# B&R Automation Studio project Parker_BMM_ST_V5_3147_V12 (part 27)

#### alarm.c
```c
/********************************************************************
 * COPYRIGHT --  B&R China
 ********************************************************************
 * Program: gAlarm
 * File: gAlarm.c
 * Author: lijianjun
 * Created: March 06, 2013
 ********************************************************************
 * Implementation of program gAlarm --- gAlarm and gImply control
 ********************************************************************/

#include <bur/plctypes.h>
#include <string.h>

#ifdef _DEFAULT_INCLUDES
#include <AsDefault.h>
#endif

#include "defines.h"
#include "edge.h"
#include "keyap2100.h"
//#include "keyap880.h"
#include "pic_id.h"

/* gAlarm text display mode  */
#define	 S$ALARM_TEXT_TOP	      0
#define	 S$ALARM_TEXT_LIST	   1

/**************************************************************************************
** 			       function ALARM type -- warning or alarm  				  			    **
**************************************************************************************/
void AlarmTyp(Alarm_typ * pInst);

/**************************************************************************************
     	        		I N I T U P  O F   T H E   T A S K
**************************************************************************************/
_INIT void alarm_init ( void )
{
	memset(AlarmBit,0,sizeof(AlarmBit));
	memset(OldPBit ,0,sizeof(OldPBit));
	memset(OldNBit ,0,sizeof(OldNBit));

	memset(&gImply,0,sizeof(gImply));

	AlarmCount = 0;
	TimeCounter  = 30;
	iFunction = 1;

	memset(&AlarmBand,1,sizeof(AlarmBand));
	AlarmTyp(&AlarmBand);

}

/**************************************************************************************
        				C Y C L I C   P A R T   O F   T H E   T A S K
**************************************************************************************/

_CYCLIC void alarm_cyclic ( void )
{
	int i,j;
	if(TimeCounter > 0)
	{
		memset(&gAlarm,0,sizeof(gAlarm));
		memset(&LMold.Alarm,0,sizeof(LMold.Alarm));
		memset(&RMold.Alarm,0,sizeof(RMold.Alarm));

		TimeCounter--;
		return;
	}

	pAlarmband = (USINT *)(&AlarmBand);

	gAlarm.batteryLow     = ap880Battery;
	gAlarm.EmergencyStop  = gMachineIn.InstancyStop;

	IsHeat = 0;
	for (i = 0; i<MAX_IDX_CONTRL_ZONES;i++)
	{
		if (1 == gT_Par.Ctl.OnOff[i])
		{
			IsHeat = 1;
			break;
		}
	}

	if(1 == gT_Par.Status.bLow)
	{
		gMachineInfo.ExtrTLow = 1;
		if(1 == IsHeat)
		{
			gAlarm.ScrewTempLow = 1;
		}
		else
		{
			gAlarm.ScrewTempLow = 0;
		}
	}
	else
	{
		gMachineInfo.ExtrTLow = 0;
		gAlarm.ScrewTempLow   = 0;
	}

	gAlarm.ScrewTempHigh	     = gT_Par.Status.bHigh;
	//	if (1==gAlarm.ScrewTempHigh)
	//	{
	//		gMachineOut.HeatPower=0;
	//	}

	if (1==gAlarm.HeatError)
	{
		gMachineOut.HeatPower=0;
	}

	gAlarm.TempFanErr		= gMachineIn.TempFanErr;
	gAlarm.ThermocoupleBroken = gT_Par.Status.bBroken;
	gAlarm.OilPumpFilter  = !gMachineIn.OilPumpFilter ;
	gAlarm.CoolingPumpFilter = !gMachineIn.CoolingPumpFilter;
	gAlarm.TonnageFilter = !gMachineIn.TonnagePumpFilter;
	gAlarm.PneuForceNormal = !gMachineIn.PneuForceNormal ;

	gAlarm.HeatingPowerNormal = !gMachineIn.HeatingPowerNormal;

	gAlarm.OilPumpErr = gMachineIn.OilPumpErr;
//	gAlarm.AirPressureLow = !gMachineIn.LMold.AirPressureLow || !gMachineIn.RMold.AirPressureLow;
	/*20180926 ipis*/
	gAlarm.OilPump1Overload = gMachineIn.OilPump1Overload;
	gAlarm.OilPump2Overload = gMachineIn.OilPump2Overload;
	gAlarm.ParisonMotorOverload = gMachineIn.ParisonPumpMotorErr;
	gAlarm.PlateMotorOverload = gMachineIn.PlateMotorOverload;

	gAlarm.WaterPressureLow = gMachineIn.WaterPressureLow;

	/* -------------- 風壓異常 延時 ----------------*/
	if (1 == gMachineInfo.Auto) //ipis0924
	{
		//		gAlarm.AirPressureLow = gMachineIn.AirPressureLow ;

		if( gMachineIn.LMold.AirPressureLow || gMachineIn.RMold.AirPressureLow)  //owen 20201027
		{
			gMacTimer.AirPressureLowAlarmDly.IN = 1;
			gMacTimer.AirPressureLowAlarmDly.PT = gUserFix_new.AirPressureLowAlarmDlyTime;
			gAlarm.AirPressureLowDly = 1;
			if(1 == gMacTimer.AirPressureLowAlarmDly.Q)
			{
				gAlarm.AirPressureLow = 1;
				gAlarm.AirPressureLowDly = 0;
				gMacTimer.AirPressureLowAlarmDly.IN = 0;
				gMachineInfo.AirPressureLowDlyFlag = 1;
			}

			switch (AirPressureLowStatus)
			{
				case 0:
					gMacTimer.AirPressureLowAlarmDly.IN = 1;
					gMacTimer.AirPressureLowAlarmDly.PT = gUserFix_new.AirPressureLowAlarmDlyTime;
					gAlarm.AirPressureLowDly = 1;
					if(1 == gMacTimer.AirPressureLowAlarmDly.Q)
					{
						gMacTimer.AirPressureLowAlarmDly.IN = 0;
						gAlarm.AirPressureLowDly = 0;
						gAlarm.AirPressureLow = 1;
						gMachineInfo.AirPressureLowDlyFlag = 1;
						StatusDelay = 2;
						AirPressureLowStatus = 10;
					}
					break;
				case 10:
					AlarmSound = 1;
					if(StatusDelay > 0 )StatusDelay--;
					if( 0 == StatusDelay)
					{
						AirPressureLowStatus = 20;
					}
					//reset

					break;
				case 20:

					break;

			}

		}
		else
		{
			gMacTimer.AirPressureLowAlarmDly.IN = 0;
			gAlarm.AirPressureLowDly  = 0;
			AirPressureLowStatus = 0;
		}
	}
	else
	{
		AirPressureLowStatus = 0;
	}

	gAlarm.Voltage24vNormal = !gMachineIn.Voltage24vNormal;
	gAlarm.L_LubricNormal = !gMachineIn.LMold.LubricNormal;
	gAlarm.R_LubricNormal = !gMachineIn.RMold.LubricNormal;

//	if(1 == LMold.Option.RobotTransfer)
//	{
//		gAlarm.ServoTransferErrL = LMold.Robot.Transfer.Error;
//		gAlarm.ServoTransProtectL = LMold.Robot.Transfer.BwHWSwitch | LMold.Robot.Transfer.FwHWSwitch;
//	}
//	else
//	{
//		gAlarm.ServoTransferErrL = 0;
//		gAlarm.ServoTransProtectL = 0;
//	}

	if(1 == LMold.Option.RobotUpDn)
	{
		gAlarm.ServoUpDnErrL = LMold.Robot.UpDn.Error;
		gAlarm.ServoUpDnProtectL  = LMold.Robot.UpDn.BwHWSwitch | LMold.Robot.UpDn.FwHWSwitch;
	}
	else
	{
		gAlarm.ServoUpDnErrL = 0;
		gAlarm.ServoUpDnProtectL = 0;
	}

//	if(1 == RMold.Option.RobotTransfer)
//	{
//		gAlarm.ServoTransferErrR = RMold.Robot.Transfer.Error;
//		gAlarm.ServoTransProtectR = RMold.Robot.Transfer.BwHWSwitch | RMold.Robot.Transfer.FwHWSwitch;
//	}
//	else
//	{
//		gAlarm.ServoTransferErrR = 0;
//		gAlarm.ServoTransProtectR = 0;
//	}

	if(1 == RMold.Option.RobotUpDn)
	{
		gAlarm.ServoUpDnErrR = RMold.Robot.UpDn.Error;
		gAlarm.ServoUpDnProtectR  = RMold.Robot.UpDn.BwHWSwitch | RMold.Robot.UpDn.FwHWSwitch;
	}
	else
	{
		gAlarm.ServoUpDnErrR = 0;
		gAlarm.ServoUpDnProtectR =0;
	}

	gMachineIn.LMold.CarriageLockLimit = ! LMold.Option.Enable;
	if(LMold.Option.Enable == gMachineIn.LMold.CarriageLockLimit)
	{
		gAlarm.CarriageLockL = 1;
	}
	else
	{
		gAlarm.CarriageLockL = 0;
	}

	gMachineIn.RMold.CarriageLockLimit = ! RMold.Option.Enable;
	if(RMold.Option.Enable == gMachineIn.RMold.CarriageLockLimit)
	{
		gAlarm.CarriageLockR = 1;
	}
	else
	{
		gAlarm.CarriageLockR = 0;
	}

	gAlarm.ModuleErr = gPROCESS_info.moduleErr;

	gAlarm.OilPosition = !gMachineIn.OilPositionNormal;

	gAlarm.LubriFilter   = gMachineIn.LubriFilter;
	gAlarm.LubriOverload = gMachineIn.LubriOverload;

	if(0 == gMachineFix.OilCooling.OilTempAlarm)  gMachineFix.OilCooling.OilTempAlarm = 40;
	if(gMachineInfo.OilTemp > gMachineFix.OilCooling.OilTempAlarm)
	{
		gAlarm.OilTempHigh = 1;
	}
	else
	{
		gAlarm.OilTempHigh = 0;
	}

	if(gServoLinear.Current > -32767 && gServoLinear.Current < 32767)
	{
		gAlarm.ParisonLinearBreak = 0;
	}
	else
	{
		gAlarm.ParisonLinearBreak = 1;
	}

	memcpy(&gAlarm.LAlarm,&LMold.Alarm,sizeof(gAlarm.LAlarm));
	memcpy(&gAlarm.RAlarm,&RMold.Alarm,sizeof(gAlarm.RAlarm));

	memcpy(&gAlarm.LHwAlarm,&LMold.HwAlarm,sizeof(gAlarm.LHwAlarm));
	memcpy(&gAlarm.RHwAlarm,&RMold.HwAlarm,sizeof(gAlarm.RHwAlarm));

	memcpy(AlarmBit,&gAlarm,sizeof(gAlarm));

	IsAlarm   = 0;
	IsWarning = 0;

	/* ------------------------ 当前报警 ----------------------------- */

	for(i=0;i<sizeof(gAlarm);i++)
	{
		if(1 == EDGEPOS(AlarmBit[i],OldPBit[i]))
		{
			gMachineInfo.AlarmIndex = i+1;
			if(1 == pAlarmband[i])
			{
				AlarmSound = 1;
			}
		}
		else if((1 == EDGENEG(AlarmBit[i],OldNBit[i]))&&(0 == gAlarm.EmergencyStop))
		{
			gMachineInfo.AlarmIndex  = 0;
			AlarmSound = 0;
		}
		else
		{
			if(1 == AlarmBit[i])
			{
				gMachineInfo.AlarmIndex = i+1;
			}
		}

		OldPBit[i] = AlarmBit[i];
		OldNBit[i] = AlarmBit[i];

		if(1 == AlarmBit[i])
		{
			if(1 == pAlarmband[i])
			{
				IsAlarm = 1;
			}
			else
			{
				IsWarning = 1;
			}
		}
	}/* for(i=0;i<sizeof(gAlarm);i++) */

	AlarmCount ++;

	/* ------------------------- 警报闪动图标 ---------------------------- */
	if(1 == IsAlarm || 1 == IsWarning)
	{
		if((AlarmCount%10) < 5)
		{
			gMachineInfo.IsAlarm = 1;
		}
		else
		{
			gMachineInfo.IsAlarm = 0;
		}
	}
	else
	{
		gMachineInfo.IsAlarm = 0;
	}

	/* ------------------------- 输出警报文字 ---------------------------- */
	if (gPanelObj.vcHandle == 0)
	{

	}
	else if (IsAlarm || IsWarning)
	{
		if((AlarmCount%3) == 0)
		{
			if (!VA_Saccess (1, gPanelObj.vcHandle))
			{
				if(iFunction > 2 || iFunction < 1)iFunction = 1;
				AlarmLength = sizeof(sAlarmText)/sizeof(sAlarmText[0]);
				Status_wcGetAlarmList = VA_wcGetActAlarmList(1, gPanelObj.vcHandle, (UDINT)sAlarmTmp, (UDINT)&AlarmLength, iFunction, '|', 2);

				if (Status_wcGetAlarmList == 240)
				{
					iFunction = 1;
					lengthTotal = record;
					record = 0;
					memcpy(sAlarmTotal,sAlarmTotalTmp,sizeof(sAlarmTotalTmp));
				}
				else if(Status_wcGetAlarmList == 0)
				{
					if(S$ALARM_TEXT_TOP == gMachineFix.Option.AlarmTextMode )
						{
						iFunction = 1;
					}
					else
					{
						iFunction = 2;
					}

					if(iFunctionOld == 1 && iFunction == 2)
					{
						memset(sAlarmTotalTmp,0,sizeof(sAlarmTotalTmp));
					}

					j = 0;
					for(i=0;i<sizeof(sAlarmText)/sizeof(sAlarmText[0]);i++)
					{
						if(sAlarmTmp[i] == '|')
						{
							IndexArray[j] = i;
							j++;
						}

						if(sAlarmTmp[i] == 0)
						{
							break;
						}
					}/* for(i=0;i<sizeof(sAlarmText)/sizeof(sAlarmText[0]);i++) */

					memset(sAlarmText,0,sizeof(sAlarmText));
					if(IndexArray[3] > IndexArray[2] + 2)
					{
						for(i=IndexArray[2]+1;i<IndexArray[3];i++)
						{
							sAlarmText[i - IndexArray[2] - 1] = sAlarmTmp[i];
							if(record < 180)
							{
								sAlarmTotalTmp[record + i - IndexArray[2] - 1] = sAlarmTmp[i];
							}
						}

						sAlarmTmp[IndexArray[3] - IndexArray[2] - 1] = 0;

						if(record < 180)
						{
							sAlarmTotalTmp[record + IndexArray[3] - IndexArray[2] - 1] = '/';
							record = record + IndexArray[3] - IndexArray[2];
						}
					}/* if(IndexArray[1] > IndexArray[2] + 2) */
				}/* else if(Status_wcGetAlarmList == 0) */
				VA_Srelease (1, gPanelObj.vcHandle);
			}/* if (!VA_Saccess (1, vcHandle)) */
		}/* if((AlarmCount%3) == 0) */
	}
	else  /* else if (IsAlarm) */
	{
		memset(sAlarmText,0,sizeof(sAlarmText));
	}/* if (vcHandle == 0) */

	iFunctionOld = iFunction;

	/* ------------ gAlarm led mode ----------- */

	if (1 == IsAlarm )
	{
		if( 1 == gAlarm.AirPressureLowDly )
		{
			gMachineInfo.AlarmLight.Red = 0;
			gMachineInfo.AlarmLight.Yellow = 1;
			gMachineInfo.AlarmLight.Green = 0;
		}
		else
		{
			gMachineInfo.AlarmLight.Red = 1;
			gMachineInfo.AlarmLight.Yellow = 0;
			gMachineInfo.AlarmLight.Green = 0;
		}
	}
	else
	{
		gMachineInfo.AlarmLight.Red = 0;
		if(1 == gMachineInfo.IsImply ||  (1 == gExtruderTempLow_HMIFlag && 1 == gMachineOut.HeatPower) ) // 加溫啟動 但溫度未到（與壓出機啟動條件相同）
		{
			gMachineInfo.AlarmLight.Yellow = 1;
			gMachineInfo.AlarmLight.Green = 0;
		}
		else
		{
			gMachineInfo.AlarmLight.Yellow = 0;
			gMachineInfo.AlarmLight.Green = 1;
		}

	}

	gMachineOut.AlarmRed 	= gMachineInfo.AlarmLight.Red;
	gMachineOut.AlarmYellow = gMachineInfo.AlarmLight.Yellow;
	gMachineOut.AlarmGreen 	= gMachineInfo.AlarmLight.Green;

	//	if(0 == gMachineFix.Option.AlarmLedMode)
	//	{
	//		gMachineOut.AlarmRed = IsAlarm;
	//	}
	//	else
	//	{
	//		gMachineOut.AlarmRed = gMachineInfo.IsAlarm;
	//	}

	//	gMachineOut.AlarmYellow = IsWarning;

	/* ------------ gAlarm sound mode ----------- */

	if(1 == AlarmSound)
	{
//		if((AlarmCount%8) < 4)
//		{
//			gMachineOut.AlarmBuzzer = 1;
//		}
//		else
//		{
//			gMachineOut.AlarmBuzzer = 0;
//		}

		//Alarm Buzzer Echo Mode
		AlarmBuzzerCount ++;
		if((AlarmBuzzerCount < 5))
		{
			gMachineOut.AlarmBuzzer = 1;
		}
		else
		{
			if(AlarmBuzzerCount > 7) AlarmBuzzerCount = 0;
			gMachineOut.AlarmBuzzer = 0;
		}

//		gMachineOut.AlarmBuzzer = 1;

	}
	else
	{
		gMachineOut.AlarmBuzzer  = 0;
		AlarmBuzzerCount = 0;
	}
	/* ------------------------ 消除报警 -------------------------------- */
	if(1 == EDGEPOS(gPanelObj.KeyMatric[S$KEYMATRIX_ALARM_RESET],OldAlarmConfirmOK))
	{
		memset(&gAlarm,0,sizeof(gAlarm));
		memset(&LMold.Alarm,0,sizeof(LMold.Alarm));
		memset(&RMold.Alarm,0,sizeof(RMold.Alarm));
		memset(&LMold.HwAlarm,0,sizeof(LMold.HwAlarm));
		memset(&RMold.HwAlarm,0,sizeof(RMold.HwAlarm));
		/*gExtruderACtrl.InverterCmd.bResetFault = 1*/
	}

	if(1 == gPanelObj.KeyMatric[S$KEYMATRIX_ALARM_RESET])
	{
		AlarmSound = 0;
		gPROCESS_info.extruderStopEnable = 0;
	}
	OldAlarmConfirmOK = gPanelObj.KeyMatric[S$KEYMATRIX_ALARM_RESET];

	/*Albert P84 Error reset by Visual Key*/
	gExtruderACtrl.InverterCmd.bResetFault = gPanelObj.KeyMatric[S$KEYMATRIX_ALARM_RESET];
	gExtruderBCtrl.InverterCmd.bResetFault = gPanelObj.KeyMatric[S$KEYMATRIX_ALARM_RESET];
	gExtruderCCtrl.InverterCmd.bResetFault = gPanelObj.KeyMatric[S$KEYMATRIX_ALARM_RESET];
	gExtruderVCtrl.InverterCmd.bResetFault = gPanelObj.KeyMatric[S$KEYMATRIX_ALARM_RESET];

		/* ------------------------- 系统提示信息  ------------------------- */
		for(i=0;i<sizeof(gImply);i++)
	{
		if((1 == ((USINT *)&gImply)[i]  ) &&
			(0 == ((USINT*)&OldImply)[i]))    /* edge positive */
		{
			gMachineInfo.ImplyTime  = 51;     /*  10 second gImply time */
			gMachineInfo.IsImply    = 1;
			gMachineInfo.ImplyIdex  = i + 1;
		}
		((USINT *)&OldImply)[i] = (( USINT *)&gImply)[i];
	}

	if(gMachineInfo.ImplyTime > 0)
	{
		gMachineInfo.ImplyTime --;
	}

	if(1 == gMachineInfo.ImplyTime)
	{
		memset(&gImply,0,sizeof(gImply));

		gMachineInfo.IsImply   = 0;
		gMachineInfo.ImplyIdex = 0;
	}

	for(i=0;i<32;i++)
	{
		if(1 == gPanelObj.KeyMatric[i] )
		{
			if(1 == gMachineInfo.Manual || 1 == gMachineInfo.Calib )
			{
				if ( 1 == gMachineInfo.IsImply ) gMachineOut.ImplyBuzzer  = 1;
			}
		}

//		if(1 == EDGEPOS(gPanelObj.KeyMatric[i],PKeyMatric[i]) )
//		{
//			if(1 == gMachineInfo.Manual || 1 == gMachineInfo.Calib )
//			{
//				if ( 1 == gMachineInfo.IsImply ) gMachineOut.ImplyBuzzer  = 1;
//			}
//
//		}

		if(1 ==  EDGENEG(gPanelObj.KeyMatric[i],NKeyMatric[i]) )
		{
			gMachineOut.ImplyBuzzer  = 0;
			gMachineInfo.ImplyTime = 2 ;
		}
	}
}/* task end */

void AlarmTyp(Alarm_typ * pInst)
{
	pInst->batteryLow     = 0;
	pInst->ModuleErr      = 1;
	pInst->SaftyDoor      = 1;
	pInst->EmergencyStop  = 1;

	pInst->ScrewTempLow   = 0;
	pInst->ScrewTempHigh  = 0;
	pInst->ThermocoupleBroken = 1;
	pInst->TempException      = 1;

	pInst->OilPumpErr      = 1;
	pInst->CoolingPumpErr  = 0;
	pInst->VisuExtrMotorOverload = 1;
	pInst->A_ExtruderMotorOverload = 1;
	pInst->B_ExtruderMotorOverload = 1;

	pInst->ParisonLinearBreak   = 1;
	pInst->ParisonLinearCalErr  = 1;
	pInst->ParisonValuebeyond   = 0;
	pInst->OilPumpFilter        = 0;

	memset(&pInst->LAlarm,1,sizeof(pInst->LAlarm));
	memset(&pInst->RAlarm,1,sizeof(pInst->RAlarm));
//	pInst->LAlarm.ParisonTimeSmall = 0;
//	pInst->RAlarm.ParisonTimeSmall = 0;

	pInst->LCycleTime = 1;
	pInst->RCycleTime = 1;

	pInst->OilPosition  = 0;
	pInst->LubrTimeZero    = 0;

	pInst->OilTempHigh = 0;
	pInst->OilPumpOff  = 1;

	pInst->LCarriageLinearBreak = 1;
	pInst->RCarriageLinearBreak = 1;
	pInst->LClampLinearBreak = 1;
	pInst->RClampLinearBreak = 1;

	pInst->LowSafeValvePumpOff = 1;
	pInst->HighSafeValvePumpOff = 1;
	pInst->LubriFilter   = 0;
	pInst->LubriOverload = 0;

	pInst->VisuExtrCoolOverload = 0;
	pInst->CoolingPumpErr  = 0;
	pInst->AccuSensorError  = 1;
	pInst->AccuChargeError  = 1;

	pInst->ExtrAMeltP_Alarm  = 1;
	pInst->ExtrBMeltP_Alarm = 1;
	pInst->ExtrACurrentAlarm  = 1;
	pInst->ExtrBCurrentAlarm = 1;
	pInst->A_ExtrMotorOverload =1;
	pInst->B_ExtrMotorOverload =1;
	pInst->C_ExtrMotorOverload =1;
	pInst->V_ExtrMotorOverload =1;

	pInst->HeatError=1;

	pInst->AccuChargeRPressure =1;
	pInst->AirPressureLow = 1;
	pInst->AirPressureLowDly = 1;
	pInst->OilTempHigh	= 1;

	pInst->AirPressureLow=1; //ipis0924
	pInst->WaterPressureLow=1;//ipis0924

}/*  void AlarmTyp(Alarm_typ * pInst) */
```

#### alarm.var
```iecst
VAR
	AlarmBit : ARRAY[0..MAX_ALARM_NUM] OF BOOL;
	AlarmBand : Alarm_typ;
	pAlarmband : REFERENCE TO USINT;
	iFunctionOld : UINT;
	iFunction : UINT;
	Status_wcGetAlarmList : UINT;
	AlarmLength : UINT;
	lengthTotal : UINT;
	record : UINT;
	TimeCounter : UDINT;
	AlarmSound : USINT;
	ImplySound : USINT;
	IsAlarm : USINT;
	IsWarning : USINT;
	OldImply : Imply_typ;
	OldPBit : ARRAY[0..MAX_ALARM_NUM] OF USINT;
	OldNBit : ARRAY[0..MAX_ALARM_NUM] OF USINT;
	OldAlarmConfirmOK : USINT;
	IsHeat : USINT;
	AlarmCount : UDINT;
	ap880Battery : USINT;
	IndexArray : ARRAY[0..9] OF UINT;
	sAlarmText : ARRAY[0..MAX_ALARM_TEXT] OF UINT;
	sAlarmTmp : ARRAY[0..MAX_ALARM_TEXT] OF UINT;
	sAlarmTotalTmp : ARRAY[0..199] OF UINT := [200(0)];
	sAlarmTotal : ARRAY[0..199] OF UINT;
	PKeyMatric : ARRAY[0..MAX_KEY_COUNT] OF USINT;
	NKeyMatric : ARRAY[0..MAX_KEY_COUNT] OF USINT;
	AirPressureLowStatus : UINT;
	StatusDelay : USINT;
	AlarmBuzzerCount : USINT;
END_VAR
```

- pic_id.h (reference to Logical/GlobalIncludes/pic_id.h)

- defines.h (reference to Logical/GlobalIncludes/defines.h)

- keyap880.h (reference to Logical/GlobalIncludes/keyap880.h)

### Program Logical/machine/energy (ANSIC)

#### Variables.var
```iecst
VAR
	tTask : REAL := 0.0;
	RTInfo_v : RTInfo;
	cntRunTime : UDINT;
	tEnergyTime_1 : REAL;
	tEnergyTimeDis_1 : REAL;
	tEnergyTime_2 : REAL;
	tEnergyTimeDis_2 : REAL;
	AvgEnergyOld : REAL;
	AvgEnergyHeatingOld : REAL;
	tEnergyTime_3 : REAL;
	tEnergyTimeDis_3 : REAL;
	AvgEnergyPumpOld : REAL;
END_VAR
```

#### Main.c
```c
#include <bur/plctypes.h>

#ifdef _DEFAULT_INCLUDES
	#include <AsDefault.h>
#endif

void _INIT ProgramInit(void)
{
	// Insert code here
	RTInfo_v.enable = 1;
	RTInfo(&RTInfo_v);
	tTask  = RTInfo_v.cycle_time/1000.0/1000.0;

	tEnergyTime_1 = 0.0;
	tEnergyTime_2 = 0.0;

	cntRunTime = 0;

}

void _CYCLIC ProgramCyclic(void)
{
	// Insert code here
	UDINT  Temp;

	/* ---------------------------- Energy monitor ------------------------- */
	if(gUserPara.SetTimePower < 1)gUserPara.SetTimePower = 10;
	Temp  = (UDINT)(gUserPara.SetTimePower * 60 / tTask);

	if(1 == gMachineInfo.Auto)
	{
		if(cntRunTime >= Temp * 100 )cntRunTime = 0;
		if(0 == (cntRunTime % Temp))
		{
//			gMachineInfo.AvgEnergy = (gMachineInfo.AenergyT_1 - AvgEnergyOld) * 60.0 /gUserPara.SetTimePower;
//			gMachineInfo.AvgEnergyHeating = (gMachineInfo.AenergyT_2 - AvgEnergyHeatingOld)* 60.0 /gUserPara.SetTimePower;

			gMachineInfo.EnergyInfo[0].AvgEnergy = (gMachineInfo.EnergyInfo[0].AenergyT - AvgEnergyOld) * 60.0 /gUserPara.SetTimePower;/*Albert*/
			gMachineInfo.EnergyInfo[1].AvgEnergy = (gMachineInfo.EnergyInfo[1].AenergyT - AvgEnergyHeatingOld)* 60.0 /gUserPara.SetTimePower;/*Albert*/
			gMachineInfo.EnergyInfo[2].AvgEnergy = (gMachineInfo.EnergyInfo[2].AenergyT - AvgEnergyPumpOld) * 60.0/gUserPara.SetTimePower;/*Albert*/

//			AvgEnergyOld = gMachineInfo.AenergyT_1 ;
//			AvgEnergyHeatingOld = gMachineInfo.AenergyT_2 ;

			AvgEnergyOld = gMachineInfo.EnergyInfo[0].AenergyT;
			AvgEnergyHeatingOld = gMachineInfo.EnergyInfo[1].AenergyT;
			AvgEnergyPumpOld = gMachineInfo.EnergyInfo[2].AenergyT;/*Albert for pump consumption*/
		}
		cntRunTime = cntRunTime + 1;
	}
	else
	{
		cntRunTime = 0;
	}

	/* First AP3131 Old*/
	if(1 == gHardWare.AP3131_1.ClearEnergy)
	{
		tEnergyTime_1 = 0.0;
		AvgEnergyOld = 0;/*Albert*/
	}
	else
	{
		tEnergyTime_1 = tEnergyTime_1 + tTask;
	}

	tEnergyTimeDis_1 = tEnergyTime_1/60.0;

	gHardWare.AP3131_1.EnableEnergy = 1;
	if(gUserPara.Current32767_A < 1.0)gUserPara.Current32767_A = 300.0;
	gUserPara.Power32767_A   = 4.0;

	gMachineInfo.Current_A1 = gHardWare.AP3131_1.IrmsA * gUserPara.Current32767_A/1000.0/50.0;
	gMachineInfo.Current_B1 = gHardWare.AP3131_1.IrmsB * gUserPara.Current32767_A/1000.0/50.0;
	gMachineInfo.Current_C1 = gHardWare.AP3131_1.IrmsC * gUserPara.Current32767_A/1000.0/50.0;
	gMachineInfo.Power_1    = gHardWare.AP3131_1.PmeanT * gUserPara.Power32767_A/1000.0;
	gMachineInfo.AenergyT_1 = gHardWare.AP3131_1.AenergyT * gUserPara.Current32767_A/1000.0/50.0;
	gMachineInfo.SumAenergyT_1 = gHardWare.AP3131_1.SAenergyT * gUserPara.Current32767_A/1000.0/50.0;

	/*First AP3131 New*/

	gMachineInfo.EnergyInfo[0].Current_A = gHardWare.AP3131_1.IrmsA * gUserPara.Current32767_A/1000.0/50.0;
	gMachineInfo.EnergyInfo[0].Current_B = gHardWare.AP3131_1.IrmsB * gUserPara.Current32767_A/1000.0/50.0;
	gMachineInfo.EnergyInfo[0].Current_C = gHardWare.AP3131_1.IrmsC * gUserPara.Current32767_A/1000.0/50.0;
	gMachineInfo.EnergyInfo[0].Power    = gHardWare.AP3131_1.PmeanT * gUserPara.Power32767_A/1000.0;
	gMachineInfo.EnergyInfo[0].AenergyT = gHardWare.AP3131_1.AenergyT * gUserPara.Current32767_A/1000.0/50.0;
	gMachineInfo.EnergyInfo[0].SumAenergyT = gHardWare.AP3131_1.SAenergyT * gUserPara.Current32767_A/1000.0/50.0;

	/* Second AP3131 old */
	if(1 == gHardWare.AP3131_2.ClearEnergy)
	{
		tEnergyTime_2 = 0.0;
		AvgEnergyHeatingOld = 0; /*Albert*/
	}
	else
	{
		tEnergyTime_2 = tEnergyTime_2 + tTask;
	}

	tEnergyTimeDis_2 = tEnergyTime_2/60.0;

	gHardWare.AP3131_2.EnableEnergy = 1;
	if(gUserPara.Current32767_B < 1.0)gUserPara.Current32767_B = 100.0;
	gUserPara.Power32767_B = 4.0;

	gMachineInfo.Current_A2 = gHardWare.AP3131_2.IrmsA * gUserPara.Current32767_B/1000.0/50.0;
	gMachineInfo.Current_B2 = gHardWare.AP3131_2.IrmsB * gUserPara.Current32767_B/1000.0/50.0;
	gMachineInfo.Current_C2 = gHardWare.AP3131_2.IrmsC * gUserPara.Current32767_B/1000.0/50.0;
	gMachineInfo.Power_2    = gHardWare.AP3131_2.PmeanT * gUserPara.Power32767_B/1000.0;
	gMachineInfo.AenergyT_2 = gHardWare.AP3131_2.AenergyT * gUserPara.Current32767_B/1000.0/50.0;
	gMachineInfo.SumAenergyT_2 = gHardWare.AP3131_2.SAenergyT * gUserPara.Current32767_B/1000.0/50.0;

	/* Second AP3131 New*/

	gMachineInfo.EnergyInfo[1].Current_A = gHardWare.AP3131_2.IrmsA * gUserPara.Current32767_B/1000.0/50.0;
	gMachineInfo.EnergyInfo[1].Current_B = gHardWare.AP3131_2.IrmsB * gUserPara.Current32767_B/1000.0/50.0;
	gMachineInfo.EnergyInfo[1].Current_C = gHardWare.AP3131_2.IrmsC * gUserPara.Current32767_B/1000.0/50.0;
	gMachineInfo.EnergyInfo[1].Power    = gHardWare.AP3131_2.PmeanT * gUserPara.Power32767_B/1000.0;
	gMachineInfo.EnergyInfo[1].AenergyT = gHardWare.AP3131_2.AenergyT * gUserPara.Current32767_B/1000.0/50.0;
	gMachineInfo.EnergyInfo[1].SumAenergyT = gHardWare.AP3131_2.SAenergyT * gUserPara.Current32767_B/1000.0/50.0;

	/* Third AP3131 */
	if(1 == gHardWare.AP3131_3.ClearEnergy)
	{
		tEnergyTime_3 = 0.0;
		AvgEnergyPumpOld = 0;/*Albert*/
	}
	else
	{
		tEnergyTime_3 = tEnergyTime_3 + tTask;
	}

	tEnergyTimeDis_3 = tEnergyTime_3/60.0;

	gHardWare.AP3131_3.EnableEnergy = 1;
	if(gUserPara.Current32767_C < 1.0)gUserPara.Current32767_C = 100.0;
	gUserPara.Power32767_C = 4.0;

	gMachineInfo.EnergyInfo[2].Current_A = gHardWare.AP3131_3.IrmsA * gUserPara.Current32767_C/1000.0/50.0;
	gMachineInfo.EnergyInfo[2].Current_B = gHardWare.AP3131_3.IrmsB * gUserPara.Current32767_C/1000.0/50.0;
	gMachineInfo.EnergyInfo[2].Current_C = gHardWare.AP3131_3.IrmsC * gUserPara.Current32767_C/1000.0/50.0;
	gMachineInfo.EnergyInfo[2].Power    = gHardWare.AP3131_3.PmeanT * gUserPara.Power32767_C/1000.0;
	gMachineInfo.EnergyInfo[2].AenergyT = gHardWare.AP3131_3.AenergyT * gUserPara.Current32767_C/1000.0/50.0;
	gMachineInfo.EnergyInfo[2].SumAenergyT = gHardWare.AP3131_3.SAenergyT * gUserPara.Current32767_C/1000.0/50.0;
}

void _EXIT ProgramExit(void)
{
	// Insert code here

}
```

### Program Logical/machine/extru_plk (ANSIC)

#### extru_plk.c - Init, cyclic, exit code
```c
/*********************************************************************************
 * Copyright: B&R China Ningbo
 * Author:    wangz
 * Created:   May 29, 2017/10:52 AM
 *********************************************************************************/

#include <bur/plctypes.h>
#include <string.h>

#ifdef _DEFAULT_INCLUDES
#include <AsDefault.h>
#endif

/**************************************************************************************
** 					               include user files								          **
**************************************************************************************/
#include "edge.h"               /*edge function                         */
#include "keyap2100.h"
#include "pic_id.h"

/**************************************************************************************
** 					 	                 define								                   **
**************************************************************************************/
#define     S$EXTRUDER_WAIT		            	0
#define     S$EXTRUDER_CONTACTOR_ON		      	10
#define     S$EXTRUDER_POWER_ON_DELAY		  	20
#define     S$EXTRUDER_POWER_ON		         	30
#define     S$EXTRUDER_READY		            100
#define     S$EXTRUDER_BASIC_ZONE		      	110
#define     S$EXTRUDER_PRODUCTION_ZONE	      	130
#define     S$EXTRUDER_DEC_ZONE		         	150
#define     S$EXTRUDER_POWER_OFF_DECEL		   	200
#define     S$EXTRUDER_POWER_OFF_PROTECT	   	210
#define     S$EXTRUDER_POWER_OFF_DELAY		   	220
/**************************************************************************************
                               Function Declarations
**************************************************************************************/
void SpeedUpDw(short ins_des,short command,speedAdjust_typ * pSpeedUpDwData);

void ExtruderCtrl(Extruder_Ctrl_typ * pExtruder,Extruder_Para_typ * pExtrPara,speedAdjust_typ * pSpeedUpDwData);

/**************************************************************************************
     	        	       I N I T U P  O F   T H E   T A S K
**************************************************************************************/
void _INIT extru_plkINIT(void)
{
	/* TODO: Add code here */
	RTInfo_Task.enable = 1;
	RTInfo(&RTInfo_Task);

	tTask = RTInfo_Task.cycle_time/1000.0/1000.0;		/*  from us ---> s  */

	MotorSpeedA.minVal  	  = 0;
	MotorSpeedA.frequence	  = 30;
	MotorSpeedA.waitTimeSlow = 200;
	MotorSpeedA.waitTimeFast = 500;
	MotorSpeedA.unitsSlow    = 1;
	MotorSpeedA.unitsFast	= 5;
	MotorSpeedA.unitsVFast	= 20;

	MotorSpeedA.maxVal = 1000;
	MotorSpeedA.minVal = 0;

	MotorSpeedB.minVal  	 = 0;
	MotorSpeedB.frequence	 = 30;
	MotorSpeedB.waitTimeSlow = 200;
	MotorSpeedB.waitTimeFast = 500;
	MotorSpeedB.unitsSlow    = 1;
	MotorSpeedB.unitsFast	 = 5;
	MotorSpeedB.unitsVFast	 = 20;

	MotorSpeedB.maxVal = 1000;
	MotorSpeedB.minVal = 0;

	MotorSpeedVisu.frequence	= 30;
	MotorSpeedVisu.waitTimeSlow = 200;
	MotorSpeedVisu.waitTimeFast = 500;
	MotorSpeedVisu.unitsSlow    = 1;
	MotorSpeedVisu.unitsFast	= 5;
	MotorSpeedVisu.unitsVFast	= 20;

	MotorSpeedVisu.maxVal = 1000;
	MotorSpeedVisu.minVal = 0;

	cntExtruderStopDelay = 0;

	gExtruderA.Step = S$EXTRUDER_WAIT;
	gExtruderB.Step = S$EXTRUDER_WAIT;
	gExtruderVisu.Step = S$EXTRUDER_WAIT;

	gExtruderA.tTask  = tTask;
	gExtruderB.tTask  = tTask;
	gExtruderVisu.tTask = tTask;

	bHideExtrB = 0;
	bHideExtrV = 1;

	/*Ramp Function*/

	gExtruderACtrl.InverterFub.fnLCRRamp.enable = 1;
	gExtruderACtrl.InverterFub.fnLCRRamp.dy_up = 100.0;
	gExtruderACtrl.InverterFub.fnLCRRamp.dy_down = 200.0;
	gExtruderACtrl.InverterFub.fnLCRRamp.y_max = 20000.0;
	gExtruderACtrl.InverterFub.fnLCRRamp.y_min = -20000.0;
	gExtruderACtrl.InverterFub.fnLCRRamp.set = 0.0;
	gExtruderACtrl.InverterFub.fnLCRRamp.y_set = 0;

	/*Albert, give set speed value*/
//	gExtruderACtrl.SetSpeed =	ExtruderA_Retain.SetExtrSpeed * ExtruderA_Retain.Pro;
//	gExtruderBCtrl.SetSpeed =	ExtruderB_Retain.SetExtrSpeed * ExtruderB_Retain.Pro;
//	gExtruderCCtrl.SetSpeed =	ExtruderC_Retain.SetExtrSpeed * ExtruderC_Retain.Pro;
//	gExtruderVCtrl.SetSpeed =	ExtruderV_Retain.SetExtrSpeed * ExtruderV_Retain.Pro;

}
/**************************************************************************************
        				   C Y C L I C   P A R T   O F   T H E   T A S K
**************************************************************************************/
void _CYCLIC extru_plkCYCLIC(void)
{
	/*Command All control*/

	if(EnableAll_HMI)
	{
		EnableA_HMI = 1;
		EnableB_HMI = 1;
		EnableC_HMI = 1;
		EnableV_HMI = 1;
		EnableAll_HMI = 0;
	}

	if(1==DisableAll_HMI || 1==gMachineInfo.CycleTimeCounReach)
	{
		EnableA_HMI = 0;
		EnableB_HMI = 0;
		EnableC_HMI = 0;
		EnableV_HMI = 0;
		DisableAll_HMI = 0;
		gMachineInfo.CycleTimeCounReach=0;
	}

	if ( 0==gExtruderACtrl.InverterCmd.bSwitchOn)	//ipis0213
	{
		if (1== EnableA_HMI)
		{
			gImply.ExtruderA_NotOn =1;
			EnableA_HMI=0;
		}
	}
	if ( 0==gExtruderBCtrl.InverterCmd.bSwitchOn)	//ipis0213
	{
		if (1== EnableB_HMI)
		{
			gImply.ExtruderB_NotOn =1;
			EnableB_HMI=0;
		}
	}
	if ( 0==gExtruderCCtrl.InverterCmd.bSwitchOn)	//ipis0213
	{
		if (1== EnableC_HMI)
		{
			gImply.ExtruderC_NotOn =1;
			EnableC_HMI=0;
		}
	}
	if ( 0==gExtruderVCtrl.InverterCmd.bSwitchOn)	//ipis0213
	{
		if (1== EnableV_HMI)
		{
			gImply.ExtruderV_NotOn =1;
			EnableV_HMI=0;
		}
	}

	/*--------------------------------------------------------------*/
	/*----------------------Extruder A------------------------------*/
	/*--------------------------------------------------------------*/
//	if(gExtruderACtrl.InverterStatus.PowerOnReady == 1)
//	{
		gMachineOut.ExtrA_Power = gExtruderACtrl.InverterCmd.bSwitchOn;				// For extruder A fan

	if(1 == EDGEPOS(gPanelObj.KeyMatric[S$KEYMATRIX_EXTRUDER_A_PLK],PKeyMatric[S$KEYMATRIX_EXTRUDER_A_PLK]))
		{
		if (0==gExtruderTempLow_HMIFlag)  //ipis0719
		{
			if (0==gMachineInfo.bLoweringFlag)
			{
				gImply.TempLow = gMachineInfo.ExtrTLow;
				gImply.HeaterPowerNotOn = !gMachineOut.HeatPower;
				gImply.HeatNotOn=!gT_Par.GrpSwh.OnOff[0];
				gMachineOut.ExtrA_Enable =!gMachineOut.ExtrA_Enable;

				gExtruderACtrl.InverterCmd.bEnableCtrl = !gExtruderACtrl.InverterCmd.bEnableCtrl; //ipis1214
				gExtruderACtrl.InverterCmd.bSwitchOn = !gExtruderACtrl.InverterCmd.bSwitchOn;

			}
			else
			{
				gImply.TempLoweringEnable =1;
			}
		}
		else
		{
		gImply.TempLow =1;

		}
	}

		if (gMachineInfo.ExtrTLow 	 || gAlarm.TempException	|| /*memcmp(&gAlarm.LAlarm, &null, sizeof(gAlarm.LAlarm)) != 0 ||*/
			/*gAlarm.AlarmExtrMeltP 	 ||*/ /*gAlarm.WarnExtrMeltP 	||*/
			gAlarm.A_BarrelCoolFault || gAlarm.A_ExtrCoolFault 		|| gAlarm.ThermocoupleBroken ||
			/*gAlarm.CarriageAxisError ||*/ /*gAlarm.LCarriageLinearBreak ||*/ /*gAlarm.LClampLinearBreak ||*/ /*gAlarm.ParisonLinearBreak ||*/
			gAlarm.EmergencyStop || (0 == gMachineOut.HeatPower) /*||  (0 == gMachineInfo.IsHeat)*/ /*|| 0==gAlarm.A_ExtrMotorOverload*/|| 0==gT_Par.GrpSwh.OnOff[0] )
		{
			EnableA_HMI = 0;
		gMachineOut.ExtrA_Enable=0;
		//	gExtruderACtrl.InverterCmd.bSwitchOn = 0;
		gExtruderACtrl.InverterCmd.bEnableCtrl = 0; //ipis1214
		gExtruderACtrl.InverterCmd.bSwitchOn = 0;
		}

//		if(gExtruderACtrl.InverterStatus.bSwitchOn == 1)
//		{
///////////////////////////////////////////////////////////////////////////	ipis 1214
//			if(EnableA_HMI == 1)
//			{
//				gExtruderACtrl.InverterCmd.bEnableCtrl = 1;
//			gExtruderACtrl.InverterCmd.bSwitchOn = 1;//
//
//			}
//			else
//			{
//				gExtruderACtrl.InverterCmd.bEnableCtrl = 0;
//		gExtruderACtrl.InverterCmd.bSwitchOn = 0;//
//			}
/////////////////////////////////////////////////////////////////////////////////////
//		}
//		else
//		{
//			EnableA_HMI = 0;
//			gExtruderACtrl.InverterCmd.bEnableCtrl  = 0;
//		}
//	}
	if (0==gMachineOut.ExtrA_Enable)
	{
		EnableA_HMI = 0;
	}
	if(gExtruderACtrl.InverterStatus.bSwitchOn == 1)
	{
		gAlarm.A_ExtrMotorOverload = gMachineIn.ExtrA_MotorErr;
		if (1==gAlarm.A_ExtrMotorOverload)
		{
			EnableA_HMI = 0;
			EnableB_HMI = 0;
			EnableC_HMI = 0;
			EnableV_HMI = 0;

		//	gExtruderACtrl.InverterCmd.bSwitchOn = 0;
			gMachineOut.ExtrA_Enable=0;
			gMachineOut.ExtrB_Enable=0;
			gMachineOut.ExtrC_Enable=0;
			gMachineOut.ExtrV_Enable=0;
		}
	}

	/*--------------------------------------------------------------*/
	/*----------------------Extruder B------------------------------*/
	/*--------------------------------------------------------------*/
//	if(gExtruderBCtrl.InverterStatus.PowerOnReady == 1)
//	{
		gMachineOut.ExtrB_Power = gExtruderBCtrl.InverterCmd.bSwitchOn;				// For extruder B fan

	if(1 == EDGEPOS(gPanelObj.KeyMatric[S$KEYMATRIX_EXTRUDER_B_PLK],PKeyMatric[S$KEYMATRIX_EXTRUDER_B_PLK]))
		{
		if (0==gExtruderTempLow_HMIFlag) //ipis0719
		{
			if (0==gMachineInfo.bLoweringFlag)
			{
				gImply.TempLow = gMachineInfo.ExtrTLow;
				gImply.HeaterPowerNotOn = !gMachineOut.HeatPower;
				gImply.HeatNotOn=!gT_Par.GrpSwh.OnOff[0];
				gMachineOut.ExtrB_Enable =!gMachineOut.ExtrB_Enable;

				gExtruderBCtrl.InverterCmd.bEnableCtrl = !gExtruderBCtrl.InverterCmd.bEnableCtrl;  //ipis1214
				gExtruderBCtrl.InverterCmd.bSwitchOn	=!gExtruderBCtrl.InverterCmd.bSwitchOn;
			}
			else
			{
				gImply.TempLoweringEnable =1;
			}
		}
		else
		{
			gImply.TempLow =1;

		}

	}

		if (gMachineInfo.ExtrTLow 	 || gAlarm.TempException	|| /*memcmp(&gAlarm.LAlarm, &null, sizeof(gAlarm.LAlarm)) != 0 ||*/
			/*gAlarm.AlarmExtrMeltP 	 ||*/ /*gAlarm.WarnExtrMeltP 	||*/
			gAlarm.B_BarrelCoolFault || gAlarm.B_ExtrCoolFault 		|| gAlarm.ThermocoupleBroken ||
			/*gAlarm.CarriageAxisError ||*/ /*gAlarm.LCarriageLinearBreak ||*/ /*gAlarm.LClampLinearBreak ||*/ /*gAlarm.ParisonLinearBreak ||*/
			gAlarm.EmergencyStop || (0 == gMachineOut.HeatPower) /*||  (0 == gMachineInfo.IsHeat)*/ /*|| 0==gAlarm.B_ExtrMotorOverload*/|| 0==gT_Par.GrpSwh.OnOff[0] )
		{
			EnableB_HMI = 0;
		gMachineOut.ExtrB_Enable=0;
		gExtruderBCtrl.InverterCmd.bEnableCtrl = 0;  //ipis1214
		gExtruderBCtrl.InverterCmd.bSwitchOn	=0;
		}

	//	if(gExtruderBCtrl.InverterStatus.bSwitchOn == 1)
	//	{
/////////////////////////////////////////////////////////////////////////////////////
//			if(EnableB_HMI == 1)
//			{
//				gExtruderBCtrl.InverterCmd.bEnableCtrl = 1;
//		gExtruderBCtrl.InverterCmd.bSwitchOn=1;
//			}
//			else
//			{
//				gExtruderBCtrl.InverterCmd.bEnableCtrl = 0;
//		gExtruderBCtrl.InverterCmd.bSwitchOn=0;
//			}
////////////////////////////////////////////////////////////////////////////////////////////
	//	}
	//	else
	//	{
	//		EnableB_HMI = 0;
	//		gExtruderBCtrl.InverterCmd.bEnableCtrl  = 0;
	//	}
//	}
	if (0==gMachineOut.ExtrB_Enable)
	{
		EnableB_HMI = 0;
	}
	if(gExtruderBCtrl.InverterStatus.bSwitchOn == 1)
	{
		gAlarm.B_ExtrMotorOverload = gMachineIn.ExtrB_MotorErr;

		if (1==gAlarm.B_ExtrMotorOverload)
		{
		//	EnableB_HMI = 0;
			EnableA_HMI = 0;
			EnableB_HMI = 0;
			EnableC_HMI = 0;
			EnableV_HMI = 0;
		//	gExtruderBCtrl.InverterCmd.bSwitchOn = 0;
		//	gMachineOut.ExtrB_Enable=0;
			gMachineOut.ExtrA_Enable=0;
			gMachineOut.ExtrB_Enable=0;
			gMachineOut.ExtrC_Enable=0;
			gMachineOut.ExtrV_Enable=0;
		}
	}

	/*--------------------------------------------------------------*/
	/*----------------------Extruder C------------------------------*/
	/*--------------------------------------------------------------*/
//	if(gExtruderCCtrl.InverterStatus.PowerOnReady == 1)
//	{
		gMachineOut.ExtrC_Power = gExtruderCCtrl.InverterCmd.bSwitchOn;				// For extruder C fan

	if(1 == EDGEPOS(gPanelObj.KeyMatric[S$KEYMATRIX_EXTRUDER_C_PLK],PKeyMatric[S$KEYMATRIX_EXTRUDER_C_PLK]))
		{
		if (0==gExtruderTempLow_HMIFlag)  //ipis0719
		{
			if (0==gMachineInfo.bLoweringFlag)
			{
				gImply.TempLow = gMachineInfo.ExtrTLow;
				gImply.HeaterPowerNotOn = !gMachineOut.HeatPower;
				gImply.HeatNotOn=!gT_Par.GrpSwh.OnOff[0];
				gMachineOut.ExtrC_Enable =!gMachineOut.ExtrC_Enable;

				gExtruderCCtrl.InverterCmd.bEnableCtrl 	=	!gExtruderCCtrl.InverterCmd.bEnableCtrl;
				gExtruderCCtrl.InverterCmd.bSwitchOn	=	!gExtruderCCtrl.InverterCmd.bSwitchOn;

			}
			else
			{
				gImply.TempLoweringEnable =1;
			}
		}
		else
		{
			gImply.TempLow =1;

		}

	}

		if (gMachineInfo.ExtrTLow 	 || gAlarm.TempException	|| /*memcmp(&gAlarm.LAlarm, &null, sizeof(gAlarm.LAlarm)) != 0 ||*/
			/*gAlarm.AlarmExtrMeltP 	 ||*/ /*gAlarm.WarnExtrMeltP 	||*/
			gAlarm.C_BarrelCoolFault || gAlarm.C_ExtrCoolFault 	 	|| gAlarm.ThermocoupleBroken ||
			/*gAlarm.CarriageAxisError ||*/ /*gAlarm.LCarriageLinearBreak ||*//* gAlarm.LClampLinearBreak ||*/ /*gAlarm.ParisonLinearBreak ||*/
			gAlarm.EmergencyStop || (0 == gMachineOut.HeatPower) /*||  (0 == gMachineInfo.IsHeat)*/ /*|| 0==gAlarm.C_ExtrMotorOverload*/ || 0==gT_Par.GrpSwh.OnOff[0])
		{
			EnableC_HMI = 0;
		gMachineOut.ExtrC_Enable=0;

		gExtruderCCtrl.InverterCmd.bEnableCtrl = 0;
		gExtruderCCtrl.InverterCmd.bSwitchOn=0;
		}
	//	if(gExtruderCCtrl.InverterStatus.bSwitchOn == 1)
	//	{
////////////////////////////////////////////////////////////////////////////////////
//			if(EnableC_HMI == 1)
//			{
//				gExtruderCCtrl.InverterCmd.bEnableCtrl = 1;
//		gExtruderCCtrl.InverterCmd.bSwitchOn=1;
//			}
//			else
//			{
//				gExtruderCCtrl.InverterCmd.bEnableCtrl = 0;
//		gExtruderCCtrl.InverterCmd.bSwitchOn=0;
//			}
/////////////////////////////////////////////////////////////////////////////////////
	//	}
	//	else
	//	{
	//		EnableC_HMI = 0;
	//		gExtruderCCtrl.InverterCmd.bEnableCtrl  = 0;
	//	}
//	}
	if (0==gMachineOut.ExtrC_Enable)
	{
		EnableC_HMI = 0;
	}
	if(gExtruderCCtrl.InverterStatus.bSwitchOn == 1)
	{
		gAlarm.C_ExtrMotorOverload = gMachineIn.ExtrC_MotorErr;

		if (1==gAlarm.C_ExtrMotorOverload)
		{
		//	EnableC_HMI = 0;
			EnableA_HMI = 0;
			EnableB_HMI = 0;
			EnableC_HMI = 0;
			EnableV_HMI = 0;
		//	gExtruderCCtrl.InverterCmd.bSwitchOn = 0;
		//	gMachineOut.ExtrC_Enable=0;
			gMachineOut.ExtrA_Enable=0;
			gMachineOut.ExtrB_Enable=0;
			gMachineOut.ExtrC_Enable=0;
			gMachineOut.ExtrV_Enable=0;
		}
	}

	/*--------------------------------------------------------------*/
	/*----------------------Extruder V------------------------------*/
	/*--------------------------------------------------------------*/
//	if(gExtruderVCtrl.InverterStatus.PowerOnReady == 1)
//	{

		gMachineOut.VisuExtrPower = gExtruderVCtrl.InverterCmd.bSwitchOn;				// For extruder V fan

	if(1 == EDGEPOS(gPanelObj.KeyMatric[S$KEYMATRIX_VISU_EXTRUDER_PLK],PKeyMatric[S$KEYMATRIX_VISU_EXTRUDER_PLK]))
		{
		if (0==gExtruderTempLow_HMIFlag) //ipis0213
		{
			if (0==gMachineInfo.bLoweringFlag)
			{
				gImply.TempLow = gMachineInfo.ExtrTLow;
				gImply.HeaterPowerNotOn = !gMachineOut.HeatPower;
				gImply.HeatNotOn=!gT_Par.GrpSwh.OnOff[0];
				gMachineOut.ExtrV_Enable =!gMachineOut.ExtrV_Enable;
				//	gExtruderVCtrl.InverterCmd.bSwitchOn = !gExtruderVCtrl.InverterCmd.bSwitchOn;
				gExtruderVCtrl.InverterCmd.bEnableCtrl 	=	!gExtruderVCtrl.InverterCmd.bEnableCtrl;
				gExtruderVCtrl.InverterCmd.bSwitchOn	=	!gExtruderVCtrl.InverterCmd.bSwitchOn;
			}
			else
			{
				gImply.TempLoweringEnable =1;
			}
		}
		else
		{
			gImply.TempLow =1;

		}

	}

		if (gMachineInfo.ExtrTLow 	 || gAlarm.TempException	|| /*memcmp(&gAlarm.LAlarm, &null, sizeof(gAlarm.LAlarm)) != 0 ||*/
			/*gAlarm.AlarmExtrMeltP 	 ||*/ /*gAlarm.WarnExtrMeltP 	||*/
			gAlarm.V_BarrelCoolFault || gAlarm.V_ExtrCoolFault 		|| gAlarm.ThermocoupleBroken ||
			/*gAlarm.CarriageAxisError ||*/ /*gAlarm.LCarriageLinearBreak || gAlarm.LClampLinearBreak ||*/ /*gAlarm.ParisonLinearBreak ||*/
			gAlarm.EmergencyStop || (0 == gMachineOut.HeatPower) /*||  (0 == gMachineInfo.IsHeat)*/ /*|| 0==gAlarm.V_ExtrMotorOverload*/ || 0==gT_Par.GrpSwh.OnOff[0] )
		{
			EnableV_HMI = 0;
		gMachineOut.ExtrV_Enable=0;

		gExtruderVCtrl.InverterCmd.bEnableCtrl = 0;
		gExtruderVCtrl.InverterCmd.bSwitchOn=0;
		}

	//	if(gExtruderVCtrl.InverterStatus.bSwitchOn == 1)
	//	{
/////////////////////////////////////////////////////////////////////////////////
//			if(EnableV_HMI == 1)
//			{
//				gExtruderVCtrl.InverterCmd.bEnableCtrl = 1;
//		gExtruderVCtrl.InverterCmd.bSwitchOn=1;
//			}
//			else
//			{
//				gExtruderVCtrl.InverterCmd.bEnableCtrl = 0;
//		gExtruderVCtrl.InverterCmd.bSwitchOn=0;
//			}
///////////////////////////////////////////////////////////////////////////////////
	//	}
	//	else
	//	{
	//		EnableV_HMI = 0;
	//		gExtruderVCtrl.InverterCmd.bEnableCtrl  = 0;
	//	}
//	}
	if (0==gMachineOut.ExtrV_Enable)
	{
		EnableV_HMI = 0;
	}
	if(gExtruderVCtrl.InverterStatus.bSwitchOn == 1)
	{
		gAlarm.V_ExtrMotorOverload = gMachineIn.ExtrV_MotorErr;

		if (1==gAlarm.V_ExtrMotorOverload)
		{
		//	EnableV_HMI = 0;
			EnableA_HMI = 0;
			EnableB_HMI = 0;
			EnableC_HMI = 0;
			EnableV_HMI = 0;
		//	gExtruderVCtrl.InverterCmd.bSwitchOn = 0;
		//	gMachineOut.ExtrV_Enable=0;
			gMachineOut.ExtrA_Enable=0;
			gMachineOut.ExtrB_Enable=0;
			gMachineOut.ExtrC_Enable=0;
			gMachineOut.ExtrV_Enable=0;
		}
	}
	// Parison pump is followed by Extruder A //
//	if (gExtruderACtrl.InverterStatus.bSwitchOn)  //Chao-i 20180402
//	{
//		if (gMachineInfo.ExtrTLow == 0)
//		{
//			uParisonPumpEn = 1;
//		}
//		else
//		{
//			uParisonPumpEn = 0;
////			gMachineOut.ParisonPump = 0;
//		}
//	}
//	else
//	{
//		uParisonPumpEn = 0;
////		gMachineOut.ParisonPump = 0;
//	}

	if (ExtruderA_Retain.Pro == 0)
	{
		ExtruderA_Retain.Pro = 1;
	}
	if (ExtruderB_Retain.Pro == 0)
	{
		ExtruderB_Retain.Pro = 1;
	}
	if (ExtruderC_Retain.Pro == 0)
	{
		ExtruderC_Retain.Pro = 1;
	}
	if (ExtruderV_Retain.Pro == 0)
	{
		ExtruderV_Retain.Pro = 1;
	}
	for(Index=0 ; Index<3 ; Index++)
	{
		if (ExtruderA_Retain.AccTime[Index] == 0)
		{
			ExtruderA_Retain.AccTime[Index] = 1.0;
		}
		if (ExtruderB_Retain.AccTime[Index] == 0)
		{
			ExtruderB_Retain.AccTime[Index] = 1.0;
		}
		if (ExtruderC_Retain.AccTime[Index] == 0)
		{
			ExtruderC_Retain.AccTime[Index] = 1.0;
		}
		if (ExtruderV_Retain.AccTime[Index] == 0)
		{
			ExtruderV_Retain.AccTime[Index] = 1.0;
		}
	}

	ExtrASpeedLmt					= (int)MotorSpeedLmtA / ExtruderA_Retain.Pro;
	ExtrBSpeedLmt					= (int)MotorSpeedLmtB / ExtruderB_Retain.Pro;
	ExtrCSpeedLmt					= (int)MotorSpeedLmtC / ExtruderC_Retain.Pro;
	ExtrVSpeedLmt					= (int)MotorSpeedLmtV / ExtruderV_Retain.Pro;
	ExtruderA_Retain.ActExtrSpeed 	= (int)(ExtruderA_Retain.ActMotorSpeed / ExtruderA_Retain.Pro);
	ExtruderB_Retain.ActExtrSpeed 	= (int)(ExtruderB_Retain.ActMotorSpeed / ExtruderB_Retain.Pro);
	ExtruderC_Retain.ActExtrSpeed 	= (int)(ExtruderC_Retain.ActMotorSpeed / ExtruderC_Retain.Pro);
	ExtruderV_Retain.ActExtrSpeed 	= (int)(ExtruderV_Retain.ActMotorSpeed / ExtruderV_Retain.Pro);
	for(Index=0 ; Index<3 ; Index++)
	{
		ExtruderA_Retain.Acc[Index]		= (700.0)/ExtruderA_Retain.AccTime[Index]*tTask;//*ExtruderA_Retain.Pro;
		ExtruderB_Retain.Acc[Index]		= (700.0)/ExtruderB_Retain.AccTime[Index]*tTask;//*ExtruderB_Retain.Pro;
		ExtruderC_Retain.Acc[Index]		= (700.0)/ExtruderC_Retain.AccTime[Index]*tTask;//*ExtruderA_Retain.Pro;
		ExtruderV_Retain.Acc[Index]		= (700.0)/ExtruderV_Retain.AccTime[Index]*tTask;//*ExtruderB_Retain.Pro;

	}

	/*Exturder A*/
	/*if(ExtruderA_Retain.OperateEnable == 1)*/
//	if(1 == gExtruderACtrl.InverterCmd.bEnableCtrl)
//	{
//		if(gExtruderACtrl.SetSpeed < (ExtruderA_Retain.SetExtrSpeed * ExtruderA_Retain.Pro)-0.5)
//		{
//			if(gExtruderACtrl.SetSpeed <= 700*ExtruderA_Retain.Pro)
//			{
//				ExtruderA_Retain.SetMotorSpeedREAL += ExtruderA_Retain.Acc[0];
//				gExtruderACtrl.SetSpeed = (int)ExtruderA_Retain.SetMotorSpeedREAL;
//			}
//			else if(gExtruderACtrl.SetSpeed > 700*ExtruderA_Retain.Pro && gExtruderACtrl.SetSpeed <= 1400*ExtruderA_Retain.Pro)
//			{
//				ExtruderA_Retain.SetMotorSpeedREAL += ExtruderA_Retain.Acc[1];
//				gExtruderACtrl.SetSpeed = (int)ExtruderA_Retain.SetMotorSpeedREAL;
//			}
//			else if(gExtruderACtrl.SetSpeed > 1400*ExtruderA_Retain.Pro && gExtruderACtrl.SetSpeed <= 2100*ExtruderA_Retain.Pro)
//			{
//				ExtruderA_Retain.SetMotorSpeedREAL += ExtruderA_Retain.Acc[2];
//				gExtruderACtrl.SetSpeed = (int)ExtruderA_Retain.SetMotorSpeedREAL;
//			}
//		}
//		else if(gExtruderACtrl.SetSpeed > (ExtruderA_Retain.SetExtrSpeed * ExtruderA_Retain.Pro)+0.5)
//		{
//			if(gExtruderACtrl.SetSpeed <= 700*ExtruderA_Retain.Pro)
//			{
//				ExtruderA_Retain.SetMotorSpeedREAL -= ExtruderA_Retain.Acc[0];
//				gExtruderACtrl.SetSpeed = (int)ExtruderA_Retain.SetMotorSpeedREAL;
//			}
//			else if(gExtruderACtrl.SetSpeed > 700*ExtruderA_Retain.Pro && gExtruderACtrl.SetSpeed <= 1400*ExtruderA_Retain.Pro)
//			{
//				ExtruderA_Retain.SetMotorSpeedREAL -= ExtruderA_Retain.Acc[1];
//				gExtruderACtrl.SetSpeed = (int)ExtruderA_Retain.SetMotorSpeedREAL;
//			}
//			else if(gExtruderACtrl.SetSpeed > 1400*ExtruderA_Retain.Pro && gExtruderACtrl.SetSpeed <= 2100*ExtruderA_Retain.Pro)
//			{
//				ExtruderA_Retain.SetMotorSpeedREAL -= ExtruderA_Retain.Acc[2];
//				gExtruderACtrl.SetSpeed = (int)ExtruderA_Retain.SetMotorSpeedREAL;
//			}
//		}
//	}
//	else
//	{
//		ExtruderA_Retain.SetMotorSpeedREAL = 0;
//		gExtruderACtrl.SetSpeed = 0;
//	}

	/*Exturder B*/
//	if(1 == gExtruderBCtrl.InverterCmd.bEnableCtrl)
//	{
//		if(gExtruderBCtrl.SetSpeed < (ExtruderB_Retain.SetExtrSpeed * ExtruderB_Retain.Pro)-0.5)
//		{
//			if(gExtruderBCtrl.SetSpeed <= 700*ExtruderB_Retain.Pro)
//			{
//				ExtruderB_Retain.SetMotorSpeedREAL += ExtruderB_Retain.Acc[0];
//				gExtruderBCtrl.SetSpeed = (int)ExtruderB_Retain.SetMotorSpeedREAL;
//			}
//			else if(gExtruderBCtrl.SetSpeed > 700*ExtruderB_Retain.Pro && gExtruderBCtrl.SetSpeed <= 1400*ExtruderB_Retain.Pro)
//			{
//				ExtruderB_Retain.SetMotorSpeedREAL += ExtruderB_Retain.Acc[1];
//				gExtruderBCtrl.SetSpeed = (int)ExtruderB_Retain.SetMotorSpeedREAL;
//			}
//			else if(gExtruderBCtrl.SetSpeed > 1400*ExtruderB_Retain.Pro && gExtruderBCtrl.SetSpeed <= 2100*ExtruderB_Retain.Pro)
//			{
//				ExtruderB_Retain.SetMotorSpeedREAL += ExtruderB_Retain.Acc[2];
//				gExtruderBCtrl.SetSpeed = (int)ExtruderB_Retain.SetMotorSpeedREAL;
//			}
//		}
//		else if(gExtruderBCtrl.SetSpeed > (ExtruderB_Retain.SetExtrSpeed * ExtruderB_Retain.Pro)+0.5)
//		{
//			if(gExtruderBCtrl.SetSpeed <= 700*ExtruderB_Retain.Pro)
//			{
//				ExtruderB_Retain.SetMotorSpeedREAL -= ExtruderB_Retain.Acc[0];
//				gExtruderBCtrl.SetSpeed = (int)ExtruderB_Retain.SetMotorSpeedREAL;
//			}
//			else if(gExtruderBCtrl.SetSpeed > 700*ExtruderB_Retain.Pro && gExtruderBCtrl.SetSpeed <= 1400*ExtruderB_Retain.Pro)
//			{
//				ExtruderB_Retain.SetMotorSpeedREAL -= ExtruderB_Retain.Acc[1];
//				gExtruderBCtrl.SetSpeed = (int)ExtruderB_Retain.SetMotorSpeedREAL;
//			}
//			else if(gExtruderBCtrl.SetSpeed > 1400*ExtruderB_Retain.Pro && gExtruderBCtrl.SetSpeed <= 2100*ExtruderB_Retain.Pro)
//			{
//				ExtruderB_Retain.SetMotorSpeedREAL -= ExtruderB_Retain.Acc[2];
//				gExtruderBCtrl.SetSpeed = (int)ExtruderB_Retain.SetMotorSpeedREAL;
//			}
//		}
//	}
//	else
//	{
//		ExtruderB_Retain.SetMotorSpeedREAL = 0;
//		gExtruderBCtrl.SetSpeed = 0;
//	}

	/*Exturder C*/
//	if(1 == gExtruderCCtrl.InverterCmd.bEnableCtrl)
//	{
//		if(gExtruderCCtrl.SetSpeed < (ExtruderC_Retain.SetExtrSpeed * ExtruderC_Retain.Pro)-0.5)
//		{
//			if(gExtruderCCtrl.SetSpeed <= 700*ExtruderC_Retain.Pro)
//			{
//				ExtruderC_Retain.SetMotorSpeedREAL += ExtruderC_Retain.Acc[0];
//				gExtruderCCtrl.SetSpeed = (int)ExtruderC_Retain.SetMotorSpeedREAL;
//			}
//			else if(gExtruderCCtrl.SetSpeed > 700*ExtruderC_Retain.Pro && gExtruderCCtrl.SetSpeed <= 1400*ExtruderC_Retain.Pro)
//			{
//				ExtruderC_Retain.SetMotorSpeedREAL += ExtruderC_Retain.Acc[1];
//				gExtruderCCtrl.SetSpeed = (int)ExtruderC_Retain.SetMotorSpeedREAL;
//			}
//			else if(gExtruderCCtrl.SetSpeed > 1400*ExtruderC_Retain.Pro && gExtruderCCtrl.SetSpeed <= 2100*ExtruderC_Retain.Pro)
//			{
//				ExtruderC_Retain.SetMotorSpeedREAL += ExtruderC_Retain.Acc[2];
//				gExtruderCCtrl.SetSpeed = (int)ExtruderC_Retain.SetMotorSpeedREAL;
//			}
//		}
//		else if(gExtruderCCtrl.SetSpeed > (ExtruderC_Retain.SetExtrSpeed * ExtruderC_Retain.Pro)+0.5)
//		{
//			if(gExtruderCCtrl.SetSpeed <= 700*ExtruderC_Retain.Pro)
//			{
//				ExtruderC_Retain.SetMotorSpeedREAL -= ExtruderC_Retain.Acc[0];
//				gExtruderCCtrl.SetSpeed = (int)ExtruderC_Retain.SetMotorSpeedREAL;
//			}
//			else if(gExtruderCCtrl.SetSpeed > 700*ExtruderC_Retain.Pro && gExtruderCCtrl.SetSpeed <= 1400*ExtruderC_Retain.Pro)
//			{
//				ExtruderC_Retain.SetMotorSpeedREAL -= ExtruderC_Retain.Acc[1];
//				gExtruderCCtrl.SetSpeed = (int)ExtruderC_Retain.SetMotorSpeedREAL;
//			}
//			else if(gExtruderCCtrl.SetSpeed > 1400*ExtruderC_Retain.Pro && gExtruderCCtrl.SetSpeed <= 2100*ExtruderC_Retain.Pro)
//			{
//				ExtruderC_Retain.SetMotorSpeedREAL -= ExtruderC_Retain.Acc[2];
//				gExtruderCCtrl.SetSpeed = (int)ExtruderC_Retain.SetMotorSpeedREAL;
//			}
//		}
//	}
//	else
//	{
//		ExtruderC_Retain.SetMotorSpeedREAL = 0;
//		gExtruderCCtrl.SetSpeed = 0;
//	}

	/*Exturder V*/
//	if(1 == gExtruderVCtrl.InverterCmd.bEnableCtrl)
//	{
//		if(gExtruderVCtrl.SetSpeed < (ExtruderV_Retain.SetExtrSpeed * ExtruderV_Retain.Pro)-0.5)
//		{
//			if(gExtruderVCtrl.SetSpeed <= 700*ExtruderV_Retain.Pro)
//			{
//				ExtruderV_Retain.SetMotorSpeedREAL += ExtruderV_Retain.Acc[0];
//				gExtruderVCtrl.SetSpeed = (int)ExtruderV_Retain.SetMotorSpeedREAL;
//			}
//			else if(gExtruderVCtrl.SetSpeed > 700*ExtruderV_Retain.Pro && gExtruderVCtrl.SetSpeed <= 1400*ExtruderV_Retain.Pro)
//			{
//				ExtruderV_Retain.SetMotorSpeedREAL += ExtruderV_Retain.Acc[1];
//				gExtruderVCtrl.SetSpeed = (int)ExtruderV_Retain.SetMotorSpeedREAL;
//			}
//			else if(gExtruderVCtrl.SetSpeed > 1400*ExtruderV_Retain.Pro && gExtruderVCtrl.SetSpeed <= 2100*ExtruderV_Retain.Pro)
//			{
//				ExtruderV_Retain.SetMotorSpeedREAL += ExtruderV_Retain.Acc[2];
//				gExtruderVCtrl.SetSpeed = (int)ExtruderV_Retain.SetMotorSpeedREAL;
//			}
//		}
//		else if(gExtruderVCtrl.SetSpeed > (ExtruderV_Retain.SetExtrSpeed * ExtruderV_Retain.Pro)+0.5)
//		{
//			if(gExtruderVCtrl.SetSpeed <= 700*ExtruderV_Retain.Pro)
//			{
//				ExtruderV_Retain.SetMotorSpeedREAL -= ExtruderV_Retain.Acc[0];
//				gExtruderVCtrl.SetSpeed = (int)ExtruderV_Retain.SetMotorSpeedREAL;
//			}
//			else if(gExtruderVCtrl.SetSpeed > 700*ExtruderV_Retain.Pro && gExtruderVCtrl.SetSpeed <= 1400*ExtruderV_Retain.Pro)
//			{
//				ExtruderV_Retain.SetMotorSpeedREAL -= ExtruderV_Retain.Acc[1];
//				gExtruderVCtrl.SetSpeed = (int)ExtruderV_Retain.SetMotorSpeedREAL;
//			}
//			else if(gExtruderVCtrl.SetSpeed > 1400*ExtruderV_Retain.Pro && gExtruderVCtrl.SetSpeed <= 2100*ExtruderV_Retain.Pro)
//			{
//				ExtruderV_Retain.SetMotorSpeedREAL -= ExtruderV_Retain.Acc[2];
//				gExtruderVCtrl.SetSpeed = (int)ExtruderV_Retain.SetMotorSpeedREAL;
//			}
//		}
//	}
//	else
//	{
//		ExtruderV_Retain.SetMotorSpeedREAL = 0;
//		gExtruderVCtrl.SetSpeed = 0;
//	}

	/*Exturder A*/
	if((1 == gExtruderACtrl.InverterCmd.bEnableCtrl) && (1==EnableA_HMI))
	{
//		ExtruderA_Retain.SetExtrSpeed * ExtruderA_Retain.Pro

//		gExtruderACtrl.SetSpeed =	ExtruderA_Retain.SetExtrSpeed * ExtruderA_Retain.Pro;
//		gExtruderACtrl.SetSpeed =	ExtruderA_Retain.SetExtrSpeed;/*Change to the motor speed*/ //ipis0423
		gExtruderACtrl.SetSpeed =gUserPara.SetExtrSpeed_A;/*Change to the motor speed*/ //ipis0423
	}
	else
	{
		gExtruderACtrl.SetSpeed = 0;
	}

	/*Exturder B*/
	if(1 == gExtruderBCtrl.InverterCmd.bEnableCtrl && (1==EnableB_HMI))
	{
//		gExtruderBCtrl.SetSpeed =	ExtruderB_Retain.SetExtrSpeed * ExtruderB_Retain.Pro;
//		gExtruderBCtrl.SetSpeed =	ExtruderB_Retain.SetExtrSpeed;/*Change to the motor speed*/
		gExtruderBCtrl.SetSpeed =gUserPara.SetExtrSpeed_B;/*Change to the motor speed*/ //ipis0423
	}
	else
	{
		gExtruderBCtrl.SetSpeed = 0;
	}

	/*Exturder C*/
	if(1 == gExtruderCCtrl.InverterCmd.bEnableCtrl && (1==EnableC_HMI))
	{
//		gExtruderCCtrl.SetSpeed =	ExtruderC_Retain.SetExtrSpeed * ExtruderC_Retain.Pro;
//		gExtruderCCtrl.SetSpeed =	ExtruderC_Retain.SetExtrSpeed;
		gExtruderCCtrl.SetSpeed =gUserPara.SetExtrSpeed_C;/*Change to the motor speed*/ //ipis0423
	}
	else
	{
		gExtruderCCtrl.SetSpeed = 0;
	}

	/*Albert Add color speed depend on the extruder speed*/
	rCExtruderSpeed = gExtruderCCtrl.SetSpeed;

	if(ExtrCSpeedLmt != 0)
		gExtruderCCtrl.aoSetSpeed = (INT)(rCExtruderSpeed/ExtrCSpeedLmt * 32767);

	/*Exturder V*/
	if(1 == gExtruderVCtrl.InverterCmd.bEnableCtrl && (1==EnableV_HMI))
	{
//		gExtruderVCtrl.SetSpeed =	ExtruderV_Retain.SetExtrSpeed * ExtruderV_Retain.Pro;
//		gExtruderVCtrl.SetSpeed =	ExtruderV_Retain.SetExtrSpeed;
		gExtruderVCtrl.SetSpeed =gUserPara.SetExtrSpeed_V;/*Change to the motor speed*/ //ipis0423
	}
	else
	{
		gExtruderVCtrl.SetSpeed = 0;
	}

	if(ExtruderA_Retain.Pro != 0)
		gExtruderACtrl.rActRPM = gExtruderACtrl.SetSpeed/ExtruderA_Retain.Pro;
	if(ExtruderB_Retain.Pro != 0)
		gExtruderBCtrl.rActRPM = gExtruderBCtrl.SetSpeed/ExtruderB_Retain.Pro;
	if(ExtruderC_Retain.Pro != 0)
		gExtruderCCtrl.rActRPM = gExtruderCCtrl.SetSpeed/ExtruderC_Retain.Pro;
	if(ExtruderV_Retain.Pro != 0)
		gExtruderVCtrl.rActRPM = gExtruderVCtrl.SetSpeed/ExtruderV_Retain.Pro;
//	if (ExtruderA_Retain.InverseHmi == 1)
//	{
//		gExtruderACtrl.InverterCmd.bInverse = 1;
//	}
//	else
//	{
//		gExtruderACtrl.InverterCmd.bInverse = 0;
//	}
//	if (ExtruderB_Retain.InverseHmi == 1)
//	{
//		ExtruderB_Retain.Inverse = 1;
//	}
//	else
//	{
//		ExtruderB_Retain.Inverse = 0;
//	}
//	if (ExtruderC_Retain.InverseHmi == 1)
//	{
//		ExtruderC_Retain.Inverse = 1;
//	}
//	else
//	{
//		ExtruderC_Retain.Inverse = 0;
//	}
//
//	if (ExtruderV_Retain.InverseHmi == 1)
//	{
//		ExtruderV_Retain.Inverse = 1;
//	}
//	else
//	{
//		ExtruderV_Retain.Inverse = 0;
//	}

	// emergency stop
	if (gExtruderACtrl.InverterStatus.ActTorque*0.1 >= ExtruderA_Retain.AlarmTorque)
	{
		//gAxis04_ModuleOk = 1;
//		gExtruderACtrl.InverterCmd.bAskStop = 1;
	}
	else
	{
		//gAxis04_ModuleOk = 0;
//		gExtruderACtrl.InverterCmd.bAskStop = 0;
	}

	//emergency stop
	if (ExtruderB_Retain.ActTorque*0.1 >= ExtruderB_Retain.AlarmTorque)
	{
		//gAxis05_ModuleOk = 1;
//		ExtruderB_Retain.FastStop = 1;
	}
	else
	{
		//gAxis05_ModuleOk = 0;
//		ExtruderB_Retain.FastStop = 0;
	}

	if (ExtruderC_Retain.ActTorque*0.1 >= ExtruderC_Retain.AlarmTorque)
	{
		//gAxis05_ModuleOk = 1;
//		ExtruderC_Retain.FastStop = 1;
	}
	else
	{
		//gAxis05_ModuleOk = 0;
//		ExtruderC_Retain.FastStop = 0;
	}

	if (ExtruderV_Retain.ActTorque*0.1 >= ExtruderV_Retain.AlarmTorque)
	{
		//gAxis05_ModuleOk = 1;
//		ExtruderV_Retain.FastStop = 1;
	}
	else
	{
		//gAxis05_ModuleOk = 0;
//		ExtruderV_Retain.FastStop = 0;
	}

	if (ExtruderA_Retain.AlarmTorque == 0)
	{
		ExtruderA_Retain.AlarmTorque = 90;
	}
	if (ExtruderB_Retain.AlarmTorque == 0)
	{
		ExtruderB_Retain.AlarmTorque = 90;
	}
	if (ExtruderC_Retain.AlarmTorque == 0)
	{
		ExtruderC_Retain.AlarmTorque = 90;
	}
	if (ExtruderV_Retain.AlarmTorque == 0)
	{
		ExtruderV_Retain.AlarmTorque = 90;
	}

	/*2018.7.31 Albert*/
	/*Limit Extruder Set Speed*/

//	if(ExtruderA_Retain.SetExtrSpeed > ExtrASpeedLmt) ExtruderA_Retain.SetExtrSpeed = ExtrASpeedLmt;
//	if(ExtruderB_Retain.SetExtrSpeed > ExtrBSpeedLmt) ExtruderB_Retain.SetExtrSpeed = ExtrBSpeedLmt;
//	if(ExtruderC_Retain.SetExtrSpeed > ExtrCSpeedLmt) ExtruderC_Retain.SetExtrSpeed = ExtrCSpeedLmt;
//	if(ExtruderV_Retain.SetExtrSpeed > ExtrVSpeedLmt) ExtruderV_Retain.SetExtrSpeed = ExtrVSpeedLmt;

	if(ExtruderA_Retain.SetExtrSpeed > MotorSpeedLmtA) ExtruderA_Retain.SetExtrSpeed = MotorSpeedLmtA;
	if(ExtruderB_Retain.SetExtrSpeed > MotorSpeedLmtB) ExtruderB_Retain.SetExtrSpeed = MotorSpeedLmtB;
	if(ExtruderC_Retain.SetExtrSpeed > MotorSpeedLmtC) ExtruderC_Retain.SetExtrSpeed = MotorSpeedLmtC;
	if(ExtruderV_Retain.SetExtrSpeed > MotorSpeedLmtV) ExtruderV_Retain.SetExtrSpeed = MotorSpeedLmtV;

	if(gUserPara.SetExtrSpeed_A > MotorSpeedLmtA) gUserPara.SetExtrSpeed_A = MotorSpeedLmtA;
	if(gUserPara.SetExtrSpeed_B > MotorSpeedLmtB) gUserPara.SetExtrSpeed_B = MotorSpeedLmtB;
	if(gUserPara.SetExtrSpeed_C > MotorSpeedLmtC) gUserPara.SetExtrSpeed_C = MotorSpeedLmtC;
	if(gUserPara.SetExtrSpeed_V > MotorSpeedLmtV) gUserPara.SetExtrSpeed_V = MotorSpeedLmtV;

	LCRRamp(&gExtruderACtrl.InverterFub.fnLCRRamp);

}
/**************************************************************************************
        				   E X I T   P A R T   O F   T H E   T A S K
**************************************************************************************/
void _EXIT extru_plkEXIT(void)
{
	/* TODO: Add code here */
}
```

#### extru_plk.typ - Local data types
```iecst
TYPE
	speedAdjust_typ : 	STRUCT
		pSpeed : REFERENCE TO REAL;
		maxVal : REAL;
		minVal : REAL;
		frequence : REAL;
		waitTimeSlow : UINT;
		waitTimeFast : UINT;
		unitsSlow : REAL;
		unitsFast : REAL;
		unitsVFast : REAL;
		iSpeed : ARRAY[0..3]OF INT;
	END_STRUCT;
	ControlStep :
		( (*wzq*)
		READY_TO_SWITCH_ON,
		SWITCH_ON,
		ENABLE_OPERATE,
		SET_SPEED,
		FEEDBACK
		);
	ExtruderStatus_typ : 	STRUCT  (*wzq*)
		PowerOnReady : BOOL;
		SwitchOnReady : BOOL;
		EnableOnReady : BOOL;
	END_STRUCT;
END_TYPE
```

#### extru_plk.var - Local variables
```iecst
VAR
	uParisonPumpEn : USINT;
	tTask : REAL := 0.0;
	bHideExtrB : UINT;
	bHideExtrV : UINT;
	bHideExtrACmd : UINT;
	bHideExtrVCmd : UINT;
	bHideExtrBCmd : UINT;
	RTInfo_Task : RTInfo := (0);
	MotorSpeedA : speedAdjust_typ;
	MotorSpeedB : speedAdjust_typ;
	MotorSpeedVisu : speedAdjust_typ;
	PKeyMatric : ARRAY[0..MAX_KEY_COUNT] OF USINT;
	NKeyMatric : ARRAY[0..MAX_KEY_COUNT] OF USINT;
	cntExtruderStopDelay : UDINT;
	ExtruderAStatus : ExtruderStatus_typ;
	ExtruderBStatus : ExtruderStatus_typ;
	step : ControlStep; (*wzq*)
	EnableA_HMI : BOOL;
	EnableB_HMI : BOOL;
	EnableC_HMI : BOOL;
	EnableV_HMI : BOOL;
	Index : USINT;
END_VAR
VAR CONSTANT
	MotorSpeedLmt : INT := 1500;
END_VAR
VAR
	ExtrASpeedLmt : {REDUND_UNREPLICABLE} INT;
	ExtrBSpeedLmt : {REDUND_UNREPLICABLE} INT;
	ExtrCSpeedLmt : INT;
	ExtrVSpeedLmt : INT;
	null : {REDUND_UNREPLICABLE} Mold_Alarm_typ;
END_VAR
(*Insert your comment here.*)
VAR
	rCExtruderSpeed : REAL;
END_VAR
VAR CONSTANT
	MotorSpeedLmtA : INT := 1500;
	MotorSpeedLmtB : INT := 1500;
	MotorSpeedLmtC : INT := 1500;
	MotorSpeedLmtV : INT := 1500;
END_VAR
(*Cmd All button*)
VAR
	EnableAll_HMI : BOOL;
	DisableAll_HMI : BOOL;
END_VAR
```

### Program Logical/machine/Acs580Ctl (IEC)

#### Variables.var
```iecst
(********************************************************************

 * COPYRIGHT -- Microsoft

 ********************************************************************

 * Program: P84Ctl

 * File: Acs380Ctl.var

 * Author: HuangPengbin

 * Created: April 16,2018

 ********************************************************************

 * Local variables of program Acs380Ctl

 ********************************************************************)
VAR CONSTANT
	ALARM_BIT : USINT := 3;
END_VAR
VAR
	CycTime : UDINT;
	FaultFlg : ARRAY[0..NUM_ACS380_MINUS_ONE] OF BOOL;
	a : BOOL;
END_VAR
VAR CONSTANT
	ACS_FAULT : UINT := 50;
	ACS_RUN : UINT := 100;
	ACS_POWER_OFF : UINT := 0;
END_VAR
VAR
	AcsIndex : UINT;
	RstTimer : ARRAY[0..NUM_ACS380_MINUS_ONE] OF UDINT;
	RTInfo_0 : RTInfo;
END_VAR
VAR CONSTANT
	STATE_FAULT_RST : UINT := 100;
	STATE_FAULT_RST_WAIT : UINT := 110;
	STATE_RUN : UINT := 150;
	STATE_POWER_OFF : UINT := 50;
	STATE_WAIT_CMD : UINT := 10;
	STATE_ESTOP : UINT := 0;
END_VAR
VAR
	Step : ARRAY[0..NUM_ACS380_MINUS_ONE] OF UINT;
	EstopCon : ARRAY[0..NUM_ACS380_MINUS_ONE] OF UINT;
	StopCon : ARRAY[0..NUM_ACS380_MINUS_ONE] OF UINT;
	ReadySwitchOnCon : ARRAY[0..NUM_ACS380_MINUS_ONE] OF UINT;
	SwitchOnCon : ARRAY[0..NUM_ACS380_MINUS_ONE] OF UINT;
	OpeationEnCon : ARRAY[0..NUM_ACS380_MINUS_ONE] OF UINT;
	TempETAD : ARRAY[0..NUM_ACS380_MINUS_ONE] OF UINT;
	ActTorque : ARRAY[0..NUM_ACS380_MINUS_ONE] OF REAL;
END_VAR
VAR CONSTANT
	MotorSpeedLmtA : INT := 1500;
	MotorSpeedLmtVisu : INT := 1500;
	MotorSpeedLmtB : INT := 1500;
	MotorSpeedLmtC : INT := 1500;
	MotorSpeedLmtD : INT := 1500;
END_VAR
VAR
	Extruder_Use : ARRAY[0..NUM_ACS380_MINUS_ONE] OF UINT;
	Extruder_Enable : ARRAY[0..NUM_ACS380_MINUS_ONE] OF UINT;
END_VAR
```

#### Main.st
```iecst
(********************************************************************
 * COPYRIGHT -- Microsoft
 ********************************************************************
 * PROGRAM: Acs380Ctl
 * File: Acs380Cyclic.st
 * Author: HuangPengbin
 * Created: April 16, 2018
 ********************************************************************
 * Implementation OF PROGRAM Acs380Ctl
 ********************************************************************)

PROGRAM _INIT
	RTInfo_0.enable := 1;
	RTInfo_0();
	CycTime := RTInfo_0.cycle_time/1000;
	AcsIndex :=0;
	FOR AcsIndex := 0 TO NUM_ACS380_MINUS_ONE BY 1DO
		Step[AcsIndex] := STATE_ESTOP;
		gAcs380Ctrl.Command.AlmReset[AcsIndex] := 1;
		gAcs380Ctrl.Command.CMDD[AcsIndex] := 16#0406;    // 20190114
	END_FOR

END_PROGRAM

PROGRAM _CYCLIC

	IF (CTRL_ABB_POWERLINK = gMachineFix.ExtruderA.eCtrlType) THEN   // ABB Driver powerlink Commuication

		Extruder_Use[0] :=gMachineFix.ExtruderA.Use;
		Extruder_Use[1] :=gMachineFix.ExtruderB.Use;
		Extruder_Use[2] :=gMachineFix.ExtruderC.Use;
		Extruder_Use[3] :=gMachineFix.ExtruderD.Use;
		Extruder_Use[4] :=gMachineFix.ExtruderVisu.Use;

		(* AcsIndex :=0;*)
		FOR AcsIndex := 0 TO NUM_ACS380_MINUS_ONE BY 1 DO
			//ETAD是ACS380状态字
			TempETAD[AcsIndex] := gAcs380Ctrl.Status.ETAD[AcsIndex] AND 16#0008;
			////////////////////////////////////////////////////////////////////////////////////////////////////
			EstopCon[AcsIndex]			:= gAcs380Ctrl.Status.ETAD[AcsIndex] AND 16#028F;//16#0280,10#640
			StopCon[AcsIndex]			:= gAcs380Ctrl.Status.ETAD[AcsIndex] AND 16#023F;//16#0231,10#561
			ReadySwitchOnCon[AcsIndex] 	:= gAcs380Ctrl.Status.ETAD[AcsIndex] AND 16#023F;//16#0233,10#563
			SwitchOnCon[AcsIndex] 		:= gAcs380Ctrl.Status.ETAD[AcsIndex] AND 16#133F;//16#1337,10#4919
			////////////////////////////////////////////////////////////////////////////////////////////////////
			// Acs380 state  switch off;run;fault;
			FaultFlg[AcsIndex] := 0;
			IF  ( BIT_TST(TempETAD[AcsIndex],ALARM_BIT) OR (gAcs380Ctrl.Status.ModuleOk[AcsIndex] = 0)) THEN
				gAcs380Ctrl.Status.ActState[AcsIndex] := ACS_FAULT;
				FaultFlg[AcsIndex] := 1;
			END_IF
			IF ReadySwitchOnCon[AcsIndex] = 16#0233 OR EstopCon[AcsIndex] = 16#0280 THEN
				gAcs380Ctrl.Status.ActState[AcsIndex] := ACS_POWER_OFF;
			END_IF
			IF SwitchOnCon[AcsIndex] = 16#1337 OR SwitchOnCon[AcsIndex] = 16#1237 OR SwitchOnCon[AcsIndex] = 16#1B37 THEN
				gAcs380Ctrl.Status.ActState[AcsIndex] := ACS_RUN;
			END_IF

			IF FaultFlg[AcsIndex] = 1 THEN
				//			gWndCtrl.Alarm.ServErrNm[AcsIndex] := gAcs380Ctrl.Status.FaultNum[AcsIndex];//20151012 变频器错误号
			ELSE
				//			gWndCtrl.Alarm.ServErrNm[AcsIndex] := 0;
			END_IF
			///////////////////////////////////////////////////////////////////////////////////
			//		gWndCtrl.Status.ActState[AcsIndex] := gAcs380Ctrl.Status.ActState[AcsIndex];
			//		gAcs380Ctrl.Command.PowerOff[AcsIndex] := gWndCtrl.Command.PowerOff[AcsIndex];
			//		gAcs380Ctrl.Command.Move[AcsIndex] := gWndCtrl.Command.Move[AcsIndex];

			//---------------------------------ipis0508 for Plate---------------------------------------------------//
			//		gMachineOut.ExtrD_On	:=gMachineOut.MotionPower;
			//		IF 0=gMachineOut.MotionPower THEN
			//			gExtruderD.bKeyOff :=1;
			//		ELSE
			//			gExtruderD.bKeyOff :=0;
			//		END_IF;

			//****************************************************************************************************//
			gAcs380Ctrl.Command.PowerOn[0]:=	gMachineOut.ExtrA_On; //ExtruderA
			gAcs380Ctrl.Command.PowerOn[1]:=    gMachineOut.ExtrC_On; //ExtruderB
			gAcs380Ctrl.Command.PowerOn[2]:=    gMachineOut.ExtrB_On; //ExtruderC
			gAcs380Ctrl.Command.PowerOn[3]:=    gMachineOut.ExtrD_On; //ExtruderD= Plate follow MotionPower
			gAcs380Ctrl.Command.PowerOn[4]:=    gMachineOut.ExtrVisu_On; //ExtruderVisu

			//****************************************************************************************************//

			gAcs380Ctrl.Command.PowerOff[0] := 	gExtruderA.bKeyOff; //ExtruderA
			gAcs380Ctrl.Command.PowerOff[1] := 	gExtruderC.bKeyOff; //ExtruderC
			gAcs380Ctrl.Command.PowerOff[2] := 	gExtruderB.bKeyOff; //ExtruderB
			gAcs380Ctrl.Command.PowerOff[3] := 	gExtruderD.bKeyOff; //ExtruderD
			gAcs380Ctrl.Command.PowerOff[4] := 	gExtruderVisu.bKeyOff; //ExtruderVisu
			//****************************************************************************************************//

			//*********** ExtruderD= Plate follow MotionPower **************************************************//
			//		gMachineOut.ExtrD_On	:=gMachineOut.MotionPower;
			//		IF 0=gMachineOut.MotionPower THEN
			//			gExtruderD.bKeyOff :=1;
			//		ELSE
			//			gExtruderD.bKeyOff :=0;
			//		END_IF;
			//****************************************************************************************************//

//			IF gEnableAll_HMI THEN
//
//				IF 1 = gMachineFix.ExtruderA.Use THEN
//					gExtruderHMI_Enable[0]:=1;
//				END_IF;
//				IF 1 = gMachineFix.ExtruderB.Use THEN
//					gExtruderHMI_Enable[1]:=1;
//				END_IF;
//				IF 1 = gMachineFix.ExtruderC.Use THEN
//					gExtruderHMI_Enable[2]:=1;
//				END_IF;
//				IF 1 = gMachineFix.ExtruderD.Use THEN
//					gExtruderHMI_Enable[3]:=1;
//				END_IF;
//				IF 1 = gMachineFix.ExtruderVisu.Use THEN
//					gExtruderHMI_Enable[4]:=1;
//				END_IF;
//
//				gEnableAll_HMI :=0;
//			END_IF;
//
//			IF gDisableAll_HMI
//				OR 1 = gMachineIn.ExtrA_MotorErr OR 1 = gMachineIn.ExtrB_MotorErr
//				OR 1 = gMachineIn.ExtrC_MotorErr OR 1 = gMachineIn.ExtrV_MotorErr  THEN //ipis0323
//				//	gExtruderHMI_Enable[AcsIndex]:=0;
//				gExtruderHMI_Enable[0]:=0;
//				gExtruderHMI_Enable[1]:=0;
//				gExtruderHMI_Enable[2]:=0;
//				gExtruderHMI_Enable[3]:=0;
//				gExtruderHMI_Enable[4]:=0;
//
//				gDisableAll_HMI :=0;
//			END_IF;
			//****************************************************************************************************//

			gAcs380Ctrl.Command.Move[AcsIndex] := gExtruderHMI_Enable[AcsIndex];

			IF 0= AcsIndex  THEN //ExtruderA
				IF 1=Extruder_Use[AcsIndex] THEN
					// error
					IF gAcs380Ctrl.Status.FaultNum[AcsIndex] <>0 THEN
						gMachineIn.ExtrA_MotorErr :=1;
					ELSE
						gMachineIn.ExtrA_MotorErr :=0;
					END_IF;

					// Imply power not on
					IF 0=gAcs380Ctrl.Command.PowerOn[AcsIndex] THEN
						IF 1=gExtruderHMI_Enable[AcsIndex] THEN
							gImply.ExtruderA_NotOn := 1;
							gExtruderHMI_Enable[AcsIndex] :=0;
						END_IF;
					END_IF;

					// SetSpd condition
					IF (1=gExtruderHMI_Enable[AcsIndex]) AND (STATE_RUN =Step[AcsIndex]) AND (1= gAcs380Ctrl.Command.PowerOn[AcsIndex])  THEN
						gAcs380Ctrl.Command.SetSpd[AcsIndex] :=REAL_TO_INT( INT_TO_REAL((gMachinePara.ExtruderA.SetSpeed))*(20000/gMachineFix.ExtruderA.RPM10v)); //rpm //abb unit = speed : 20000  0 //ipis0718
					ELSE
						gAcs380Ctrl.Command.SetSpd[AcsIndex] := 0;
					END_IF;

					// motor speed
					gExtruderA.ActRPM := gAcs380Ctrl.Status.ActSpd[AcsIndex]*(gMachineFix.ExtruderA.RPM10v/20000);

					//Screw speed
					IF 0=gMachineFix.ExtruderA.Ratio THEN
						gMachineFix.ExtruderA.Ratio :=1;
					ELSE
						gExtruderA.ActSpeed := gExtruderA.ActRPM /gMachineFix.ExtruderA.Ratio;
					END_IF;

					//motor Current Frequency
					gExtruderA.Current_ABB := DINT_TO_REAL(gAcs380Ctrl.Status.ActCurrent[AcsIndex])/100;
					gExtruderA.Frequency_ABB := DINT_TO_REAL(gAcs380Ctrl.Status.ActFrequency[AcsIndex])/100;

				ELSE
					gExtruderHMI_Enable[AcsIndex]:=0;
					gAcs380Ctrl.Command.SetSpd[AcsIndex] := 0;
					gMachineIn.ExtrA_MotorErr :=0;
				END_IF;
			END_IF;

			IF 1= AcsIndex  THEN //ExtruderB
				IF 1=Extruder_Use[AcsIndex]  THEN
					// error
					IF gAcs380Ctrl.Status.FaultNum[AcsIndex] <>0 THEN
						gMachineIn.ExtrB_MotorErr :=1;
					ELSE
						gMachineIn.ExtrB_MotorErr :=0;
					END_IF;

					// Imply power not on
					IF 0=gAcs380Ctrl.Command.PowerOn[AcsIndex] THEN
						IF 1=gExtruderHMI_Enable[AcsIndex] THEN
							gImply.ExtruderB_NotOn := 1;
							gExtruderHMI_Enable[AcsIndex] :=0;
						END_IF;
					END_IF;

					// SetSpd condition
					IF (1=gExtruderHMI_Enable[AcsIndex]) AND (STATE_RUN =Step[AcsIndex]) AND (1= gAcs380Ctrl.Command.PowerOn[AcsIndex])  THEN
						gAcs380Ctrl.Command.SetSpd[AcsIndex] :=REAL_TO_INT( INT_TO_REAL((gMachinePara.ExtruderB.SetSpeed))*(20000/gMachineFix.ExtruderB.RPM10v)); //rpm //abb unit = speed : 20000  0 //ipis0718
					ELSE
						gAcs380Ctrl.Command.SetSpd[AcsIndex] := 0;
					END_IF;

					// motor speed
					gExtruderB.ActRPM := gAcs380Ctrl.Status.ActSpd[AcsIndex]*(gMachineFix.ExtruderB.RPM10v/20000); //ipis0620

					//Screw speed
					IF 0=gMachineFix.ExtruderB.Ratio THEN
						gMachineFix.ExtruderB.Ratio :=1;
					ELSE
						gExtruderB.ActSpeed := gExtruderB.ActRPM /gMachineFix.ExtruderB.Ratio;
					END_IF;

					//motor Current Frequency
					gExtruderB.Current_ABB := DINT_TO_REAL(gAcs380Ctrl.Status.ActCurrent[AcsIndex])/100;
					gExtruderB.Frequency_ABB := DINT_TO_REAL(gAcs380Ctrl.Status.ActFrequency[AcsIndex])/100;

				ELSE
					gExtruderHMI_Enable[AcsIndex]:=0;
					gAcs380Ctrl.Command.SetSpd[AcsIndex] := 0;
					gMachineIn.ExtrB_MotorErr :=0;
				END_IF;
			END_IF;

			IF 2= AcsIndex THEN //ExtruderC
				IF 1=Extruder_Use[AcsIndex] THEN
					// error
					IF gAcs380Ctrl.Status.FaultNum[AcsIndex] <>0 THEN
						gMachineIn.ExtrC_MotorErr :=1;
					ELSE
						gMachineIn.ExtrC_MotorErr :=0;
					END_IF;

					// Imply power not on
					IF 0=gAcs380Ctrl.Command.PowerOn[AcsIndex] THEN
						IF 1=gExtruderHMI_Enable[AcsIndex] THEN
							gImply.ExtruderC_NotOn := 1;
							gExtruderHMI_Enable[AcsIndex] :=0;
						END_IF;
					END_IF;

					// SetSpd condition
					IF (1=gExtruderHMI_Enable[AcsIndex]) AND (STATE_RUN =Step[AcsIndex]) AND (1= gAcs380Ctrl.Command.PowerOn[AcsIndex])  THEN
						gAcs380Ctrl.Command.SetSpd[AcsIndex] :=REAL_TO_INT( INT_TO_REAL((gMachinePara.ExtruderC.SetSpeed))*(20000/gMachineFix.ExtruderC.RPM10v)); //rpm //abb unit = speed : 20000  0 //ipis0718
					ELSE
						gAcs380Ctrl.Command.SetSpd[AcsIndex] := 0;
					END_IF;

					// motor speed
					gExtruderC.ActRPM := gAcs380Ctrl.Status.ActSpd[AcsIndex]*(gMachineFix.ExtruderC.RPM10v/20000); //ipis0620

					//Screw speed
					IF 0=gMachineFix.ExtruderC.Ratio THEN
						gMachineFix.ExtruderC.Ratio :=1;
					ELSE
						gExtruderC.ActSpeed := gExtruderC.ActRPM /gMachineFix.ExtruderC.Ratio;
					END_IF;

					//motor Current Frequency
					gExtruderC.Current_ABB := DINT_TO_REAL(gAcs380Ctrl.Status.ActCurrent[AcsIndex])/100;
					gExtruderC.Frequency_ABB := DINT_TO_REAL(gAcs380Ctrl.Status.ActFrequency[AcsIndex])/100;
				ELSE
					gExtruderHMI_Enable[AcsIndex]:=0;
					gAcs380Ctrl.Command.SetSpd[AcsIndex] := 0;
					gMachineIn.ExtrC_MotorErr :=0;
				END_IF;
			END_IF;

			IF 3= AcsIndex THEN //ExtruderD

				IF 1=Extruder_Use[AcsIndex]  THEN

					// error
					IF gAcs380Ctrl.Status.FaultNum[AcsIndex] <>0 THEN
						gMachineIn.ExtrD_MotorErr :=1;
					ELSE
						gMachineIn.ExtrD_MotorErr :=0;
					END_IF;

					// Imply power not on
					IF 0=gAcs380Ctrl.Command.PowerOn[AcsIndex] THEN
						IF 1=gExtruderHMI_Enable[AcsIndex] THEN
							gImply.ExtruderD_NotOn := 1;
							gExtruderHMI_Enable[AcsIndex] :=0;
						END_IF;
					END_IF;

					// SetSpd condition
					IF (1=gExtruderHMI_Enable[AcsIndex]) AND (STATE_RUN =Step[AcsIndex]) AND (1= gAcs380Ctrl.Command.PowerOn[AcsIndex])  THEN
						gAcs380Ctrl.Command.SetSpd[AcsIndex] :=REAL_TO_INT( INT_TO_REAL((gMachinePara.ExtruderD.SetSpeed))*(20000/gMachineFix.ExtruderD.RPM10v)); //rpm //abb unit = speed : 20000  0 //ipis0718
					ELSE
						gAcs380Ctrl.Command.SetSpd[AcsIndex] := 0;
					END_IF;

					// motor speed
					gExtruderD.ActRPM := gAcs380Ctrl.Status.ActSpd[AcsIndex]*(gMachineFix.ExtruderD.RPM10v/20000); //ipis0724

					//Screw speed
					IF 0=gMachineFix.ExtruderD.Ratio THEN
						gMachineFix.ExtruderD.Ratio :=1;
					ELSE
						gExtruderD.ActSpeed := gExtruderD.ActRPM /gMachineFix.ExtruderD.Ratio;
					END_IF;

					//motor Current Frequency
					gExtruderD.Current_ABB := DINT_TO_REAL(gAcs380Ctrl.Status.ActCurrent[AcsIndex])/100;
					gExtruderD.Frequency_ABB := DINT_TO_REAL(gAcs380Ctrl.Status.ActFrequency[AcsIndex])/100;

				ELSE
					gExtruderHMI_Enable[AcsIndex]:=0;
					gAcs380Ctrl.Command.SetSpd[AcsIndex] := 0;
					gMachineIn.ExtrD_MotorErr :=0;
				END_IF;
			END_IF;

			IF 4= AcsIndex THEN //ExtruderVisu

				IF 1=Extruder_Use[AcsIndex]  THEN
					// error
					IF gAcs380Ctrl.Status.FaultNum[AcsIndex] <>0 THEN
						gMachineIn.ExtrV_MotorErr :=1;
					ELSE
						gMachineIn.ExtrV_MotorErr :=0;
					END_IF;
					// Imply power not on
					IF 0=gAcs380Ctrl.Command.PowerOn[AcsIndex] THEN
						IF 1=gExtruderHMI_Enable[AcsIndex] THEN
							gImply.ExtruderV_NotOn := 1;
							gExtruderHMI_Enable[AcsIndex] :=0;
						END_IF;
					END_IF;

					IF (1=gExtruderHMI_Enable[AcsIndex]) AND (STATE_RUN =Step[AcsIndex]) AND (1= gAcs380Ctrl.Command.PowerOn[AcsIndex])  THEN
						gAcs380Ctrl.Command.SetSpd[AcsIndex] :=REAL_TO_INT( INT_TO_REAL((gMachinePara.ExtruderVisu.SetSpeed))*(20000/gMachineFix.ExtruderVisu.RPM10v)); //rpm //abb unit = speed : 20000  0 //ipis0718
					ELSE
						gAcs380Ctrl.Command.SetSpd[AcsIndex] := 0;
					END_IF;

					// motor speed
					gExtruderVisu.ActRPM := gAcs380Ctrl.Status.ActSpd[AcsIndex]*(gMachineFix.ExtruderVisu.RPM10v/20000); //ipis0620

					//Screw speed
					IF 0=gMachineFix.ExtruderVisu.Ratio THEN
						gMachineFix.ExtruderVisu.Ratio :=1;
					ELSE
						gExtruderVisu.ActSpeed := gExtruderVisu.ActRPM /gMachineFix.ExtruderVisu.Ratio;
					END_IF;

					//motor Current Frequency
					gExtruderVisu.Current_ABB := DINT_TO_REAL(gAcs380Ctrl.Status.ActCurrent[AcsIndex])/100;
					gExtruderVisu.Frequency_ABB := DINT_TO_REAL(gAcs380Ctrl.Status.ActFrequency[AcsIndex])/100;

				ELSE
					gExtruderHMI_Enable[AcsIndex]:=0;
					gAcs380Ctrl.Command.SetSpd[AcsIndex] := 0;
					gMachineIn.ExtrV_MotorErr :=0;
				END_IF;
			END_IF;

			IF (0= gAcs380Ctrl.Command.PowerOn[AcsIndex]) THEN
				Step[AcsIndex] :=STATE_ESTOP;
			END_IF;

			/////////////////////////////////////////////////////////////////////////////////////////
			CASE Step[AcsIndex] OF
				STATE_ESTOP:

					IF (1=gAcs380Ctrl.Command.PowerOn[AcsIndex] AND gAcs380Ctrl.Status.ModuleOk[AcsIndex] ) THEN // ipis0513
						IF EstopCon[AcsIndex] = 16#0280 THEN
							gAcs380Ctrl.Command.CMDD[AcsIndex] := 16#0406;
						ELSIF StopCon[AcsIndex] = 16#0231 THEN
							gAcs380Ctrl.Command.CMDD[AcsIndex] := 16#0407;
						END_IF;

						//	IF ReadySwitchOnCon[AcsIndex] = 16#0233 THEN
						Step[AcsIndex] := STATE_WAIT_CMD;
						//	END_IF;

						IF FaultFlg[AcsIndex] THEN
							gAcs380Ctrl.Command.CMDD[AcsIndex] := 16#0406; // 20190114
							Step[AcsIndex] := STATE_FAULT_RST;
						END_IF
					END_IF;

				STATE_WAIT_CMD:
					IF gAcs380Ctrl.Command.AlmReset[AcsIndex] THEN      // 20190128
						Step[AcsIndex] := STATE_FAULT_RST;
					ELSIF gAcs380Ctrl.Command.PowerOff[AcsIndex] THEN
						gAcs380Ctrl.Command.PowerOff[AcsIndex] := 0;
						Step[AcsIndex] := STATE_POWER_OFF;
					ELSIF gAcs380Ctrl.Command.Move[AcsIndex] THEN
						gAcs380Ctrl.Command.Move[AcsIndex] := 0;
						Step[AcsIndex] := STATE_RUN;
					END_IF

					IF FaultFlg[AcsIndex] THEN
						gAcs380Ctrl.Command.CMDD[AcsIndex] := 16#0406;	// 20190114
						Step[AcsIndex] := STATE_FAULT_RST;
					END_IF

				STATE_POWER_OFF:
					gAcs380Ctrl.Command.CMDD[AcsIndex] := 16#0407;
					IF ReadySwitchOnCon[AcsIndex] = 16#0233 THEN
						Step[AcsIndex] := STATE_WAIT_CMD;
					END_IF
					IF FaultFlg[AcsIndex] THEN
						gAcs380Ctrl.Command.CMDD[AcsIndex] := 16#0406;  // 20190114
						Step[AcsIndex] := STATE_FAULT_RST;
					END_IF

				STATE_FAULT_RST:
					IF  gAcs380Ctrl.Status.ModuleOk[AcsIndex] = 1 THEN
						IF BIT_TST(TempETAD[AcsIndex],ALARM_BIT) THEN
							IF gAcs380Ctrl.Command.AlmReset[AcsIndex] THEN
								gAcs380Ctrl.Command.AlmReset[AcsIndex] := 0;
								gAcs380Ctrl.Command.CMDD[AcsIndex] := 16#0080;
								Step[AcsIndex] := STATE_FAULT_RST_WAIT;
								RstTimer[AcsIndex] := 0;
							END_IF
						ELSE
							gAcs380Ctrl.Command.AlmReset[AcsIndex] := 0;
							gAcs380Ctrl.Command.CMDD[AcsIndex] := 16#0406; // 20190114
							Step[AcsIndex] := STATE_ESTOP;
						END_IF
					END_IF

				STATE_FAULT_RST_WAIT:
					RstTimer[AcsIndex] := RstTimer[AcsIndex] + CycTime;
					IF (RstTimer[AcsIndex] >= 1500) THEN
						RstTimer[AcsIndex] := 0;
						gAcs380Ctrl.Command.CMDD[AcsIndex] := 16#0406;    // 20190114
						Step[AcsIndex] := STATE_ESTOP;
					END_IF

				STATE_RUN:
					IF ReadySwitchOnCon[AcsIndex] = 16#0233 THEN
						gAcs380Ctrl.Command.CMDD[AcsIndex] := 16#040F;
					ELSIF SwitchOnCon[AcsIndex] = 16#1337 OR SwitchOnCon[AcsIndex] = 16#1237 THEN
						IF gAcs380Ctrl.Command.TorMode[AcsIndex] THEN//转距模式
							gAcs380Ctrl.Command.CMDD[AcsIndex] := 16#0C7F;
						ELSE
							gAcs380Ctrl.Command.CMDD[AcsIndex] := 16#047F;
						END_IF;
					END_IF

					IF gAcs380Ctrl.Command.PowerOff[AcsIndex] THEN
						gAcs380Ctrl.Command.PowerOff[AcsIndex] := 0;
						Step[AcsIndex] := STATE_POWER_OFF;
					END_IF

					IF FaultFlg[AcsIndex] THEN
						gAcs380Ctrl.Command.CMDD[AcsIndex] := 16#0406;    // 20190114
						Step[AcsIndex] := STATE_FAULT_RST;
					END_IF

			END_CASE

			IF FaultFlg[AcsIndex] <> 0 THEN
				gAcs380Ctrl.Status.StateIndex[AcsIndex] := 3;//错误
			END_IF;
			IF ReadySwitchOnCon[AcsIndex] = 16#0233 OR EstopCon[AcsIndex] = 16#0280 THEN
				gAcs380Ctrl.Status.StateIndex[AcsIndex] := 0;//断电
			END_IF;
			IF SwitchOnCon[AcsIndex] = 16#1337 OR SwitchOnCon[AcsIndex] = 16#1237 OR SwitchOnCon[AcsIndex] = 16#1B37 THEN
				IF gAcs380Ctrl.Status.ActSpd[AcsIndex] <> 0 THEN
					gAcs380Ctrl.Status.StateIndex[AcsIndex] := 2;//运动
				ELSE
					gAcs380Ctrl.Status.StateIndex[AcsIndex] := 1;//停止
				END_IF;
			END_IF;

			ActTorque[AcsIndex] 	:= INT_TO_REAL(gAcs380Ctrl.Status.ActTorque[AcsIndex]) / 100;

		END_FOR

	END_IF

END_PROGRAM
```

### Program Logical/machine/extruder_Mix (ANSIC, version 1.00.0) - extruder control
